# B&R Automation Studio project Teknologia25 (part 9)

#### BasicMovement.st
```iecst
ACTION BasicMoveDialGauge:
	pShuttle.function.MC_BR_MoveInPlane_Acp6D_0.Parameters.Acceleration := 5;
	pShuttle.function.MC_BR_MoveInPlane_Acp6D_0.Parameters.Velocity := 0.02;
	pShuttle.function.MC_BR_MoveInPlane_Acp6D_0.Shuttle := ADR(gAcp6DCtrl.Status.ShuttleInfo[pShuttle.par.shuttleID].shuttleRef);
	pShuttle.function.MC_BR_MoveInPlane_Acp6D_0.Parameters.Mode := 0; //Absolute
	pShuttle.function.MC_BR_MoveInPlane_Acp6D_0.Parameters.Path := 0; //direct

	CASE pShuttle.cm.state OF
		0:
			cm.description := 'Move shuttle to preDialPos';
			pShuttle.function.MC_BR_MoveInPlane_Acp6D_0.Parameters.Position.X := 0.420;
			pShuttle.function.MC_BR_MoveInPlane_Acp6D_0.Parameters.Position.Y := 0.180;
			pShuttle.function.MC_BR_MoveInPlane_Acp6D_0.Execute := TRUE;
			IF pShuttle.function.MC_BR_MoveInPlane_Acp6D_0.Acknowledge THEN
				pShuttle.function.MC_BR_MoveInPlane_Acp6D_0.Execute := FALSE;
				cm.state := 5;
			END_IF

		5:
			cm.description := 'Move shuttle to dialGauge';
			pShuttle.function.MC_BR_MoveInPlane_Acp6D_0.Parameters.Position.X := 0.420;
			pShuttle.function.MC_BR_MoveInPlane_Acp6D_0.Parameters.Position.Y := 0.190;
			pShuttle.function.MC_BR_MoveInPlane_Acp6D_0.Execute := TRUE;
			IF pShuttle.function.MC_BR_MoveInPlane_Acp6D_0.Acknowledge THEN
				pShuttle.function.MC_BR_MoveInPlane_Acp6D_0.Execute := FALSE;
				cm.state := 10;
			END_IF

		10:
			cm.description := 'Check pos reached';
			FOR i := 0 TO NUM_SHUTTLES DO
				IF((gAcp6DCtrl.Status.ShuttleInfo[pShuttle.par.shuttleID].Position.X > 0.420 - MARGIN AND gAcp6DCtrl.Status.ShuttleInfo[pShuttle.par.shuttleID].Position.X < 0.420 + MARGIN) AND
					gAcp6DCtrl.Status.ShuttleInfo[pShuttle.par.shuttleID].Position.Y > 0.190 - MARGIN AND gAcp6DCtrl.Status.ShuttleInfo[pShuttle.par.shuttleID].Position.Y < 0.190 + MARGIN) THEN
					IF gAcp6DCtrl.Status.ShuttleInfo[pShuttle.par.shuttleID].State = mcACP6D_SH_STATE_IDLING THEN
						cm.state := 20;
					END_IF
				END_IF
			END_FOR

		20:
			cm.description := 'Wait time';
			pShuttle.function.TON_0.PT := t#3s;
			pShuttle.function.TON_0.IN := TRUE;
			IF pShuttle.function.TON_0.Q THEN
				pShuttle.function.TON_0.IN := FALSE;
				cm.state := 30;
			END_IF

		30:
			cm.description := 'Move shuttle away from dialGauge';
			pShuttle.function.MC_BR_MoveInPlane_Acp6D_0.Parameters.Position.X := 0.420;
			pShuttle.function.MC_BR_MoveInPlane_Acp6D_0.Parameters.Position.Y := 0.180;
			pShuttle.function.MC_BR_MoveInPlane_Acp6D_0.Execute := TRUE;
			IF pShuttle.function.MC_BR_MoveInPlane_Acp6D_0.Acknowledge THEN
				pShuttle.function.MC_BR_MoveInPlane_Acp6D_0.Execute := FALSE;
				cm.state := 40;
			END_IF

		40:
			cm.description := 'Check pos reached';
			FOR i := 0 TO NUM_SHUTTLES DO
				IF((gAcp6DCtrl.Status.ShuttleInfo[pShuttle.par.shuttleID].Position.X > 0.420 - MARGIN AND gAcp6DCtrl.Status.ShuttleInfo[pShuttle.par.shuttleID].Position.X < 0.420 + MARGIN) AND
					gAcp6DCtrl.Status.ShuttleInfo[pShuttle.par.shuttleID].Position.Y > 0.180 - MARGIN AND gAcp6DCtrl.Status.ShuttleInfo[pShuttle.par.shuttleID].Position.Y < 0.180 + MARGIN) THEN
					IF gAcp6DCtrl.Status.ShuttleInfo[pShuttle.par.shuttleID].State = mcACP6D_SH_STATE_IDLING THEN
						cm.state := 0;
					END_IF
				END_IF
			END_FOR

	END_CASE

	cm();
	pShuttle.function.TON_0();
	pShuttle.function.MC_BR_MoveInPlane_Acp6D_0();

END_ACTION
```

#### WeightProgram.st
```iecst
ACTION weightProgram:
	pShuttle.function.MC_BR_ShGetPayload_Acp6D_0.Shuttle := ADR(gAcp6DCtrl.Status.ShuttleInfo[pShuttle.par.shuttleID].shuttleRef);

	pShuttle.function.MC_BR_MoveShortAxis_Acp6D_0.Shuttle := ADR(gAcp6DCtrl.Status.ShuttleInfo[pShuttle.par.shuttleID].shuttleRef);
	pShuttle.function.MC_BR_MoveShortAxis_Acp6D_0.Parameters.Position.Rx := 0.000;
	pShuttle.function.MC_BR_MoveShortAxis_Acp6D_0.Parameters.Position.Ry := 0.000;
	pShuttle.function.MC_BR_MoveShortAxis_Acp6D_0.Parameters.Position.Rz := 0.000;
	pShuttle.function.MC_BR_MoveShortAxis_Acp6D_0.Parameters.Position.Z := (weightProgramFlyingHight/1000); //mm to meter;
	pShuttle.function.MC_BR_MoveShortAxis_Acp6D_0.Parameters.Velocity.Z := 1;

	pShuttle.function.MC_BR_MoveInPlane_Acp6D_0.Shuttle := ADR(gAcp6DCtrl.Status.ShuttleInfo[pShuttle.par.shuttleID].shuttleRef);
	pShuttle.function.MC_BR_MoveInPlane_Acp6D_0.Parameters.Acceleration := 1;
	pShuttle.function.MC_BR_MoveInPlane_Acp6D_0.Parameters.Velocity := gAcp6DCtrl.Par.Velocity;
	pShuttle.function.MC_BR_MoveInPlane_Acp6D_0.Parameters.Path := 0; //Diagonal
	pShuttle.function.MC_BR_MoveInPlane_Acp6D_0.Parameters.Mode := 0; //absolute

	CASE cm.state OF
		0:
			cm.description := 'Move shuttle to loadLocation';
			pShuttle.function.MC_BR_MoveInPlane_Acp6D_0.Parameters.Position.X := 0.060;
			pShuttle.function.MC_BR_MoveInPlane_Acp6D_0.Parameters.Position.Y := 0.060;
			pShuttle.function.MC_BR_MoveInPlane_Acp6D_0.Execute := TRUE;
			IF pShuttle.function.MC_BR_MoveInPlane_Acp6D_0.Acknowledge THEN
				pShuttle.function.MC_BR_MoveInPlane_Acp6D_0.Execute := FALSE;
				cm.state := 5;
			END_IF

		5:
			cm.description := 'Change levitation hight';
			pShuttle.function.MC_BR_MoveShortAxis_Acp6D_0.Execute := TRUE;
			IF pShuttle.function.MC_BR_MoveShortAxis_Acp6D_0.Acknowledge THEN
				pShuttle.function.MC_BR_MoveShortAxis_Acp6D_0.Execute := FALSE;
				cm.state := 10;
			END_IF

		10:
			cm.description := 'Check pos reached';
			FOR i := 0 TO NUM_SHUTTLES DO
				IF((gAcp6DCtrl.Status.ShuttleInfo[pShuttle.par.shuttleID].Position.X > 0.060 - MARGIN AND gAcp6DCtrl.Status.ShuttleInfo[pShuttle.par.shuttleID].Position.X < 0.060 + MARGIN) AND
					gAcp6DCtrl.Status.ShuttleInfo[pShuttle.par.shuttleID].Position.Y > 0.060 - MARGIN AND gAcp6DCtrl.Status.ShuttleInfo[pShuttle.par.shuttleID].Position.Y < 0.060 + MARGIN) THEN
					IF gAcp6DCtrl.Status.ShuttleInfo[pShuttle.par.shuttleID].State = mcACP6D_SH_STATE_IDLING THEN
						cm.state := 20;
					END_IF
				END_IF
			END_FOR

		20:
			cm.description := 'Trigger robot';
			ABBRobot.startBigWeightMovement := TRUE;
			pShuttle.function.TON_0.PT := t#3s;
			pShuttle.function.TON_0.IN := TRUE;
			IF pShuttle.function.TON_0.Q THEN
				ABBRobot.startBigWeightMovement := FALSE;
				pShuttle.function.TON_0.IN := FALSE;
				cm.state := 21;
			END_IF

		21:
			cm.description := 'Calibrate weight';
			pShuttle.function.MC_BR_ShGetPayload_Acp6D_0.Execute := TRUE;
			IF pShuttle.function.MC_BR_ShGetPayload_Acp6D_0.Done THEN
				weightCalibration := pShuttle.function.MC_BR_ShGetPayload_Acp6D_0.Payload * 1000;
				pShuttle.function.MC_BR_ShGetPayload_Acp6D_0.Execute := FALSE;
				cm.state := 50;
			END_IF

//		25:
//			cm.description := 'Wait robot done';
//			IF ABBRobot.HomePositionReached THEN
//				cm.state := 50;
//			END_IF

		50:
			cm.description := 'Measure weight';
			pShuttle.function.MC_BR_ShGetPayload_Acp6D_0.Execute := TRUE;
			IF pShuttle.function.MC_BR_ShGetPayload_Acp6D_0.Done THEN
				fbPayload := pShuttle.function.MC_BR_ShGetPayload_Acp6D_0.Payload * 1000;
				shuttlePayload := fbPayload - weightCalibration;
				tempINT := REAL_TO_INT(shuttlePayload / 100);
				IF correctionValue = 0 THEN
					correctionValue := 12;
				END_IF;
				shuttlePayload := shuttlePayload - INT_TO_REAL(tempINT) * correctionValue;
				pShuttle.function.MC_BR_ShGetPayload_Acp6D_0.Execute := FALSE;
				cm.state := 60;
			END_IF

		60:
			cm.description := 'Wait time';
			pShuttle.function.TON_0.PT := t#1s;
			pShuttle.function.TON_0.IN := TRUE;
			IF pShuttle.function.TON_0.Q THEN
				pShuttle.function.TON_0.IN := FALSE;
				cm.state := 50;
			END_IF

//		80:
//			cm.description := 'Check robot ready';
//			IF ABBRobot.HomePositionReached THEN
//				ABBRobot.returnBigWeightMovement := TRUE;
//				cm.state := 81;
//			END_IF
//
//		81:
//			IF NOT ABBRobot.HomePositionReached THEN
//				ABBRobot.returnBigWeightMovement := FALSE;
//				cm.state := 90;
//			END_IF
//
//		90:
//			cm.description := 'Check when robot is done and fire small weightMovement';
//			IF ABBRobot.HomePositionReached THEN
//				ABBRobot.startSmallWeightMovement := TRUE;
//				cm.state := 100;
//			END_IF
//
//		100:
//			cm.description := 'Check robot start';
//			IF NOT ABBRobot.HomePositionReached THEN
//				ABBRobot.startSmallWeightMovement := FALSE;
//				cm.state := 110;
//			END_IF
//
//		110:
//			cm.description := 'Check robot done';
//			IF ABBRobot.HomePositionReached THEN
//				cm.state := 120;
//			END_IF
//
//		120:
//			cm.description := 'meassure small weight';
//			pShuttle.function.MC_BR_GetPayload_Acp6D_0.Execute := TRUE;
//			IF pShuttle.function.MC_BR_GetPayload_Acp6D_0.Valid THEN
//				shuttlePayload := pShuttle.function.MC_BR_GetPayload_Acp6D_0.Payload * 1000;
//				shuttlePayload := shuttlePayload - weightCalibration;
//				pShuttle.function.MC_BR_GetPayload_Acp6D_0.Execute := FALSE;
//				cm.state := 130;
//			END_IF
//
//		130:
//			cm.description := 'Wait time';
//			pShuttle.function.TON_0.PT := t#3s;
//			pShuttle.function.TON_0.IN := TRUE;
//			IF pShuttle.function.TON_0.Q THEN
//				pShuttle.function.TON_0.IN := FALSE;
//				cm.state := 140;
//			END_IF
//
//		140:
//			cm.description := 'Return small weight';
//			IF ABBRobot.HomePositionReached THEN
//				ABBRobot.returnSmallWeightMovement := TRUE;
//				cm.state := 150;
//			END_IF
//
//		150:
//			IF NOT ABBRobot.HomePositionReached THEN
//				ABBRobot.returnSmallWeightMovement := FALSE;
//				cm.state := 160;
//			END_IF
//
//		160:
//			IF ABBRobot.HomePositionReached THEN
//				modeSelector := 5; //demoProgram
//				em.cmd.sc := TRUE;
//			END_IF

	END_CASE
	pShuttle.function.MC_BR_MoveShortAxis_Acp6D_0();
	pShuttle.function.MC_BR_ShGetPayload_Acp6D_0();
	pShuttle.function.MC_BR_MoveInPlane_Acp6D_0();
	pShuttle.function.TON_0();
END_ACTION
```

#### MovementRxRyRz.st
```iecst
ACTION MovementRx:
	pShuttle.function.MC_BR_MoveShortAxis_Acp6D_0.Shuttle := ADR(gAcp6DCtrl.Status.ShuttleInfo[pShuttle.par.shuttleID].shuttleRef);
	pShuttle.function.MC_BR_MoveShortAxis_Acp6D_0.Parameters.Mode := 0; //Absolute
	pShuttle.function.MC_BR_MoveShortAxis_Acp6D_0.Parameters.Rotation.Type := 0; //Around Center
	pShuttle.function.MC_BR_MoveShortAxis_Acp6D_0.Parameters.Velocity.Rx := 0.1;
	pShuttle.function.MC_BR_MoveShortAxis_Acp6D_0.Parameters.Velocity.Rx := 0.1;
	pShuttle.function.MC_BR_MoveShortAxis_Acp6D_0.Parameters.Velocity.Ry := 0.1;
	pShuttle.function.MC_BR_MoveShortAxis_Acp6D_0.Parameters.Velocity.Z := 0.002;

	pShuttle.function.MC_BR_Move6D_Acp6D_0.Shuttle := ADR(gAcp6DCtrl.Status.ShuttleInfo[pShuttle.par.shuttleID].shuttleRef);
	CASE cm.state OF
		0:
			cm.description := 'tilt shuttle Rx';
			pShuttle.function.MC_BR_MoveShortAxis_Acp6D_0.Parameters.Position.Z := 0.002;
			pShuttle.function.MC_BR_MoveShortAxis_Acp6D_0.Parameters.Position.Rx := 0.02;
			pShuttle.function.MC_BR_MoveShortAxis_Acp6D_0.Parameters.Position.Ry := 0.00;
			pShuttle.function.MC_BR_MoveShortAxis_Acp6D_0.Parameters.Position.Rz := 0.00;
			pShuttle.function.MC_BR_MoveShortAxis_Acp6D_0.Execute := TRUE;
			IF pShuttle.function.MC_BR_MoveShortAxis_Acp6D_0.Acknowledge THEN
				pShuttle.function.MC_BR_MoveShortAxis_Acp6D_0.Execute := FALSE;
				cm.state := 10;
			ELSIF pShuttle.function.MC_BR_MoveShortAxis_Acp6D_0.Error THEN
				em.cmd.abort := TRUE;
			END_IF;

		10:
			cm.description := 'Check Rx position reached';
			IF gAcp6DCtrl.Status.ShuttleInfo[pShuttle.par.shuttleID].Position.Rx >= 0.019 THEN
				cm.state := 20;
			END_IF

		20:
			cm.description := 'tilt shuttle Rx';
			pShuttle.function.MC_BR_MoveShortAxis_Acp6D_0.Parameters.Position.Z := 0.002;
			pShuttle.function.MC_BR_MoveShortAxis_Acp6D_0.Parameters.Position.Rx := -0.02;
			pShuttle.function.MC_BR_MoveShortAxis_Acp6D_0.Parameters.Position.Ry := 0.00;
			pShuttle.function.MC_BR_MoveShortAxis_Acp6D_0.Parameters.Position.Rz := 0.00;
			pShuttle.function.MC_BR_MoveShortAxis_Acp6D_0.Execute := TRUE;
			IF pShuttle.function.MC_BR_MoveShortAxis_Acp6D_0.Acknowledge THEN
				pShuttle.function.MC_BR_MoveShortAxis_Acp6D_0.Execute := FALSE;
				cm.state := 30;
			ELSIF pShuttle.function.MC_BR_MoveShortAxis_Acp6D_0.Error THEN
				em.cmd.abort := TRUE;
			END_IF;

		30:
			cm.description := 'Check Rx position reached';
			IF gAcp6DCtrl.Status.ShuttleInfo[pShuttle.par.shuttleID].Position.Rx <= -0.019 THEN
				cm.state := 0;
			END_IF

	END_CASE

	cm();
	pShuttle.function.MC_BR_MoveShortAxis_Acp6D_0();
	pShuttle.function.MC_BR_Move6D_Acp6D_0();

END_ACTION

ACTION MovementRy:
	pShuttle.function.MC_BR_MoveShortAxis_Acp6D_0.Shuttle := ADR(gAcp6DCtrl.Status.ShuttleInfo[pShuttle.par.shuttleID].shuttleRef);
	pShuttle.function.MC_BR_MoveShortAxis_Acp6D_0.Parameters.Mode := 0; //Absolute
	pShuttle.function.MC_BR_MoveShortAxis_Acp6D_0.Parameters.Rotation.Type := 0; //Around Center
	pShuttle.function.MC_BR_MoveShortAxis_Acp6D_0.Parameters.Velocity.Rx := 0.1;
	pShuttle.function.MC_BR_MoveShortAxis_Acp6D_0.Parameters.Velocity.Rx := 0.1;
	pShuttle.function.MC_BR_MoveShortAxis_Acp6D_0.Parameters.Velocity.Ry := 0.1;
	pShuttle.function.MC_BR_MoveShortAxis_Acp6D_0.Parameters.Velocity.Z := 0.002;

	pShuttle.function.MC_BR_Move6D_Acp6D_0.Shuttle := ADR(gAcp6DCtrl.Status.ShuttleInfo[pShuttle.par.shuttleID].shuttleRef);

	CASE cm.state OF
		0:

			cm.description := 'tilt shuttle Ry';
			pShuttle.function.MC_BR_MoveShortAxis_Acp6D_0.Parameters.Position.Z := 0.002;
			pShuttle.function.MC_BR_MoveShortAxis_Acp6D_0.Parameters.Position.Ry := 0.02;
			pShuttle.function.MC_BR_MoveShortAxis_Acp6D_0.Parameters.Position.Rx := 0.00;
			pShuttle.function.MC_BR_MoveShortAxis_Acp6D_0.Parameters.Position.Rz := 0.00;
			pShuttle.function.MC_BR_MoveShortAxis_Acp6D_0.Execute := TRUE;
			IF pShuttle.function.MC_BR_MoveShortAxis_Acp6D_0.Acknowledge THEN
				pShuttle.function.MC_BR_MoveShortAxis_Acp6D_0.Execute := FALSE;
				cm.state := 10;
			ELSIF pShuttle.function.MC_BR_MoveShortAxis_Acp6D_0.Error THEN
				em.cmd.abort := TRUE;
			END_IF;

		10:
			cm.description := 'Check Rx position reached';
			IF gAcp6DCtrl.Status.ShuttleInfo[pShuttle.par.shuttleID].Position.Ry >= 0.019 THEN
				cm.state := 20;
			END_IF

		20:
			cm.description := 'tilt shuttle Ry';
			pShuttle.function.MC_BR_MoveShortAxis_Acp6D_0.Parameters.Position.Z := 0.002;
			pShuttle.function.MC_BR_MoveShortAxis_Acp6D_0.Parameters.Position.Ry := -0.02;
			pShuttle.function.MC_BR_MoveShortAxis_Acp6D_0.Parameters.Position.Rx := 0.00;
			pShuttle.function.MC_BR_MoveShortAxis_Acp6D_0.Parameters.Position.Rz := 0.00;
			pShuttle.function.MC_BR_MoveShortAxis_Acp6D_0.Execute := TRUE;
			IF pShuttle.function.MC_BR_MoveShortAxis_Acp6D_0.Acknowledge THEN
				pShuttle.function.MC_BR_MoveShortAxis_Acp6D_0.Execute := FALSE;
				cm.state := 30;
			ELSIF pShuttle.function.MC_BR_MoveShortAxis_Acp6D_0.Error THEN
				em.cmd.abort := TRUE;
			END_IF;

		30:
			cm.description := 'Check Ry position reached';
			IF gAcp6DCtrl.Status.ShuttleInfo[pShuttle.par.shuttleID].Position.Ry <= -0.019 THEN
				cm.state := 0;
			END_IF

	END_CASE

	cm();
	pShuttle.function.MC_BR_MoveShortAxis_Acp6D_0();
	pShuttle.function.MC_BR_Move6D_Acp6D_0();

END_ACTION

ACTION MovementRz:
	pShuttle.function.MC_BR_MoveShortAxis_Acp6D_0.Shuttle := ADR(gAcp6DCtrl.Status.ShuttleInfo[pShuttle.par.shuttleID].shuttleRef);
	pShuttle.function.MC_BR_MoveShortAxis_Acp6D_0.Parameters.Mode := 0; //Absolute
	pShuttle.function.MC_BR_MoveShortAxis_Acp6D_0.Parameters.Rotation.Type := 0; //Around Center
	pShuttle.function.MC_BR_MoveShortAxis_Acp6D_0.Parameters.Velocity.Rx := 0.1;
	pShuttle.function.MC_BR_MoveShortAxis_Acp6D_0.Parameters.Velocity.Rx := 0.1;
	pShuttle.function.MC_BR_MoveShortAxis_Acp6D_0.Parameters.Velocity.Ry := 0.1;
	pShuttle.function.MC_BR_MoveShortAxis_Acp6D_0.Parameters.Velocity.Z := 0.002;

	pShuttle.function.MC_BR_Move6D_Acp6D_0.Shuttle := ADR(gAcp6DCtrl.Status.ShuttleInfo[pShuttle.par.shuttleID].shuttleRef);
	CASE cm.state OF
		0:

			cm.description := 'tilt shuttle Rz';
			pShuttle.function.MC_BR_MoveShortAxis_Acp6D_0.Parameters.Position.Z := 0.002;
			pShuttle.function.MC_BR_MoveShortAxis_Acp6D_0.Parameters.Position.Rz := 0.150;
			pShuttle.function.MC_BR_MoveShortAxis_Acp6D_0.Parameters.Position.Rx := 0.00;
			pShuttle.function.MC_BR_MoveShortAxis_Acp6D_0.Parameters.Position.Ry := 0.00;
			pShuttle.function.MC_BR_MoveShortAxis_Acp6D_0.Execute := TRUE;
			IF pShuttle.function.MC_BR_MoveShortAxis_Acp6D_0.Acknowledge THEN
				pShuttle.function.MC_BR_MoveShortAxis_Acp6D_0.Execute := FALSE;
				cm.state := 10;
			ELSIF pShuttle.function.MC_BR_MoveShortAxis_Acp6D_0.Error THEN
				em.cmd.abort := TRUE;
			END_IF;

		10:
			cm.description := 'Check Rx position reached';
			IF gAcp6DCtrl.Status.ShuttleInfo[pShuttle.par.shuttleID].Position.RZ >= 0.0140 THEN
				cm.state := 20;
			END_IF

		20:
			cm.description := 'tilt shuttle Rz';
			pShuttle.function.MC_BR_MoveShortAxis_Acp6D_0.Parameters.Position.Z := 0.002;
			pShuttle.function.MC_BR_MoveShortAxis_Acp6D_0.Parameters.Position.Rz := -0.150;
			pShuttle.function.MC_BR_MoveShortAxis_Acp6D_0.Parameters.Position.Rx := 0.00;
			pShuttle.function.MC_BR_MoveShortAxis_Acp6D_0.Parameters.Position.Ry := 0.00;
			pShuttle.function.MC_BR_MoveShortAxis_Acp6D_0.Execute := TRUE;
			IF pShuttle.function.MC_BR_MoveShortAxis_Acp6D_0.Acknowledge THEN
				pShuttle.function.MC_BR_MoveShortAxis_Acp6D_0.Execute := FALSE;
				cm.state := 30;
			ELSIF pShuttle.function.MC_BR_MoveShortAxis_Acp6D_0.Aborted THEN
				em.cmd.abort := TRUE;
			END_IF;

		30:
			cm.description := 'Check Rx position reached';
			IF gAcp6DCtrl.Status.ShuttleInfo[pShuttle.par.shuttleID].Position.RZ <= -0.0140 THEN
				cm.state := 0;
			END_IF

	END_CASE

	cm();
	pShuttle.function.MC_BR_MoveShortAxis_Acp6D_0();
	pShuttle.function.MC_BR_Move6D_Acp6D_0();

END_ACTION

ACTION MovementZ:
	pShuttle.function.MC_BR_MoveShortAxis_Acp6D_0.Shuttle := ADR(gAcp6DCtrl.Status.ShuttleInfo[pShuttle.par.shuttleID].shuttleRef);
	pShuttle.function.MC_BR_MoveShortAxis_Acp6D_0.Parameters.Mode := 0; //Absolute
	pShuttle.function.MC_BR_MoveShortAxis_Acp6D_0.Parameters.Rotation.Type := 0; //Around Center
	pShuttle.function.MC_BR_MoveShortAxis_Acp6D_0.Parameters.Velocity.Rx := 0.1;
	pShuttle.function.MC_BR_MoveShortAxis_Acp6D_0.Parameters.Velocity.Rx := 0.1;
	pShuttle.function.MC_BR_MoveShortAxis_Acp6D_0.Parameters.Velocity.Ry := 0.1;
	pShuttle.function.MC_BR_MoveShortAxis_Acp6D_0.Parameters.Velocity.Z := 0.002;
	CASE em.substate OF
//		12000..12999:
//			pShuttle.function.MC_BR_MoveShortAxis_Acp6D_0.Parameters.Velocity.Z := 2;
		ELSE
			//pShuttle.function.MC_BR_MoveShortAxis_Acp6D_0.Parameters.Velocity.Z := 0.002;
			pShuttle.function.MC_BR_MoveShortAxis_Acp6D_0.Parameters.Velocity.Z := levitationVelocity;
	END_CASE
	pShuttle.function.MC_BR_Move6D_Acp6D_0.Shuttle := ADR(gAcp6DCtrl.Status.ShuttleInfo[pShuttle.par.shuttleID].shuttleRef);

	CASE cm.state OF
		0:

			cm.description := 'raise shuttle';
			pShuttle.function.MC_BR_MoveShortAxis_Acp6D_0.Parameters.Position.Z := 0.004;
			pShuttle.function.MC_BR_MoveShortAxis_Acp6D_0.Parameters.Position.Rz := 0.00;
			pShuttle.function.MC_BR_MoveShortAxis_Acp6D_0.Parameters.Position.Rx := 0.00;
			pShuttle.function.MC_BR_MoveShortAxis_Acp6D_0.Parameters.Position.Ry := 0.00;
			pShuttle.function.MC_BR_MoveShortAxis_Acp6D_0.Execute := TRUE;
			IF pShuttle.function.MC_BR_MoveShortAxis_Acp6D_0.Acknowledge THEN
				pShuttle.function.MC_BR_MoveShortAxis_Acp6D_0.Execute := FALSE;
				cm.state := 10;
			ELSIF pShuttle.function.MC_BR_MoveShortAxis_Acp6D_0.Error THEN
				em.cmd.abort := TRUE;
			END_IF;

		10:
			cm.description := 'Check Rx position reached';
			IF gAcp6DCtrl.Status.ShuttleInfo[pShuttle.par.shuttleID].Position.Z >= 0.0038 THEN
				cm.state := 20;
			END_IF

		20:
			cm.description := 'tilt shuttle Rz';
			pShuttle.function.MC_BR_MoveShortAxis_Acp6D_0.Parameters.Position.Z := 0.001;
			pShuttle.function.MC_BR_MoveShortAxis_Acp6D_0.Parameters.Position.Rz := 0.00;
			pShuttle.function.MC_BR_MoveShortAxis_Acp6D_0.Parameters.Position.Rx := 0.00;
			pShuttle.function.MC_BR_MoveShortAxis_Acp6D_0.Parameters.Position.Ry := 0.00;
			pShuttle.function.MC_BR_MoveShortAxis_Acp6D_0.Execute := TRUE;
			IF pShuttle.function.MC_BR_MoveShortAxis_Acp6D_0.Acknowledge THEN
				pShuttle.function.MC_BR_MoveShortAxis_Acp6D_0.Execute := FALSE;
				cm.state := 30;
			ELSIF pShuttle.function.MC_BR_MoveShortAxis_Acp6D_0.Error THEN
				em.cmd.abort := TRUE;
			END_IF;

		30:
			cm.description := 'Check Rz position reached';
			IF gAcp6DCtrl.Status.ShuttleInfo[pShuttle.par.shuttleID].Position.Z <= 0.0011 THEN
				cm.state := 0;
			END_IF

	END_CASE

	cm();
	pShuttle.function.MC_BR_MoveShortAxis_Acp6D_0();
	pShuttle.function.MC_BR_Move6D_Acp6D_0();
END_ACTION
```

#### linkMovement.st
```iecst
ACTION linkMovementProgram:
	//Setup
	positionContainerLinkMovement[0].Shuttle1.xPos := 0.120;
	positionContainerLinkMovement[0].Shuttle1.yPos := 0.120;
	positionContainerLinkMovement[0].Shuttle2.xPos := 0.360;
	positionContainerLinkMovement[0].Shuttle2.yPos := 0.360;
	positionContainerLinkMovement[0].Shuttle3.xPos := 0.360;
	positionContainerLinkMovement[0].Shuttle3.yPos := 0.120;
	positionContainerLinkMovement[0].Shuttle4.xPos := 0.120;
	positionContainerLinkMovement[0].Shuttle4.yPos := 0.360;

	positionContainerLinkMovement[1].Shuttle1.xPos := 0.060;
	positionContainerLinkMovement[1].Shuttle1.yPos := 0.060;
	positionContainerLinkMovement[1].Shuttle2.xPos := 0.180;
	positionContainerLinkMovement[1].Shuttle2.yPos := 0.180;
	positionContainerLinkMovement[1].Shuttle3.xPos := 0.180;
	positionContainerLinkMovement[1].Shuttle3.yPos := 0.060;
	positionContainerLinkMovement[1].Shuttle4.xPos := 0.060;
	positionContainerLinkMovement[1].Shuttle4.yPos := 0.180;

	positionContainerLinkMovement[2].Shuttle1.xPos := 0.120;
	positionContainerLinkMovement[2].Shuttle1.yPos := 0.120;
	positionContainerLinkMovement[2].Shuttle2.xPos := 0.360;
	positionContainerLinkMovement[2].Shuttle2.yPos := 0.360;
	positionContainerLinkMovement[2].Shuttle3.xPos := 0.360;
	positionContainerLinkMovement[2].Shuttle3.yPos := 0.120;
	positionContainerLinkMovement[2].Shuttle4.xPos := 0.120;
	positionContainerLinkMovement[2].Shuttle4.yPos := 0.360;

	positionContainerLinkMovement[3].Shuttle1.xPos := 0.300;
	positionContainerLinkMovement[3].Shuttle1.yPos := 0.060;
	positionContainerLinkMovement[3].Shuttle2.xPos := 0.420;
	positionContainerLinkMovement[3].Shuttle2.yPos := 0.180;
	positionContainerLinkMovement[3].Shuttle3.xPos := 0.420;
	positionContainerLinkMovement[3].Shuttle3.yPos := 0.060;
	positionContainerLinkMovement[3].Shuttle4.xPos := 0.300;
	positionContainerLinkMovement[3].Shuttle4.yPos := 0.180;

	positionContainerLinkMovement[4].Shuttle1.xPos := 0.120;
	positionContainerLinkMovement[4].Shuttle1.yPos := 0.120;
	positionContainerLinkMovement[4].Shuttle2.xPos := 0.360;
	positionContainerLinkMovement[4].Shuttle2.yPos := 0.360;
	positionContainerLinkMovement[4].Shuttle3.xPos := 0.360;
	positionContainerLinkMovement[4].Shuttle3.yPos := 0.120;
	positionContainerLinkMovement[4].Shuttle4.xPos := 0.120;
	positionContainerLinkMovement[4].Shuttle4.yPos := 0.360;

	positionContainerLinkMovement[5].Shuttle1.xPos := 0.300;
	positionContainerLinkMovement[5].Shuttle1.yPos := 0.300;
	positionContainerLinkMovement[5].Shuttle2.xPos := 0.420;
	positionContainerLinkMovement[5].Shuttle2.yPos := 0.420;
	positionContainerLinkMovement[5].Shuttle3.xPos := 0.420;
	positionContainerLinkMovement[5].Shuttle3.yPos := 0.300;
	positionContainerLinkMovement[5].Shuttle4.xPos := 0.300;
	positionContainerLinkMovement[5].Shuttle4.yPos := 0.420;

	positionContainerLinkMovement[6].Shuttle1.xPos := 0.120;
	positionContainerLinkMovement[6].Shuttle1.yPos := 0.120;
	positionContainerLinkMovement[6].Shuttle2.xPos := 0.360;
	positionContainerLinkMovement[6].Shuttle2.yPos := 0.360;
	positionContainerLinkMovement[6].Shuttle3.xPos := 0.360;
	positionContainerLinkMovement[6].Shuttle3.yPos := 0.120;
	positionContainerLinkMovement[6].Shuttle4.xPos := 0.120;
	positionContainerLinkMovement[6].Shuttle4.yPos := 0.360;

	CASE em.substate OF
		3000:
			em.description := 'Move all shuttles to prePos';
			tempShuttleCounter := 0;
			tempCounter := 0;
			em.substate := 3010;

		3010:
			em.description := 'Move all shuttles to prePos';
			IF tempShuttleCounter > NUM_SHUTTLES THEN
				tempShuttleCounter := 0;
				em.substate := 3030;
			ELSE
				MC_BR_MoveInPlane_Acp6D_0.Parameters.Acceleration := gAcp6DCtrl.Par.Acceleration;
				MC_BR_MoveInPlane_Acp6D_0.Parameters.Velocity := gAcp6DCtrl.Par.Velocity;
				MC_BR_MoveInPlane_Acp6D_0.Parameters.Mode := 0; //Abs
				MC_BR_MoveInPlane_Acp6D_0.Shuttle := ADR(gAcp6DCtrl.Status.ShuttleInfo[tempShuttleCounter].shuttleRef);
				CASE tempShuttleCounter OF
					0:
						MC_BR_MoveInPlane_Acp6D_0.Parameters.Position.X := 0.060;
						MC_BR_MoveInPlane_Acp6D_0.Parameters.Position.Y := 0.180;
					1:
						MC_BR_MoveInPlane_Acp6D_0.Parameters.Position.X := 0.180;
						MC_BR_MoveInPlane_Acp6D_0.Parameters.Position.Y := 0.180;
					2:
						MC_BR_MoveInPlane_Acp6D_0.Parameters.Position.X := 0.300;
						MC_BR_MoveInPlane_Acp6D_0.Parameters.Position.Y := 0.060;
					3:
						MC_BR_MoveInPlane_Acp6D_0.Parameters.Position.X := 0.420;
						MC_BR_MoveInPlane_Acp6D_0.Parameters.Position.Y := 0.060;
				END_CASE

				MC_BR_MoveInPlane_Acp6D_0.Execute := TRUE;
				IF MC_BR_MoveInPlane_Acp6D_0.Acknowledge THEN
					MC_BR_MoveInPlane_Acp6D_0.Execute := FALSE;
					tempShuttleCounter := tempShuttleCounter + 1;
					em.substate := 3020;
				END_IF
			END_IF

		3020:
			em.description := 'DummyScan';
			em.substate := 3010;

		3030:
			em.description := 'check shuttle state idle';
			IF gAcp6DCtrl.Status.ShuttleInfo[0].State = mcACP6D_SH_STATE_IDLING AND gAcp6DCtrl.Status.ShuttleInfo[1].State = mcACP6D_SH_STATE_IDLING
				AND gAcp6DCtrl.Status.ShuttleInfo[2].State = mcACP6D_SH_STATE_IDLING AND gAcp6DCtrl.Status.ShuttleInfo[3].State = mcACP6D_SH_STATE_IDLING AND MC_BR_AsmReadStatus_Acp6D_0.AssemblyReady THEN
				em.substate := 3035;
			END_IF

		3035:
			em.description := 'Couple ShuttleGroup1_2';
			em.cmd.sc := FALSE;
			MC_BR_ShGroupCoupleCtrl_Acp6D_0.ShuttleGroup := shGroupShuttle1_2;
			MC_BR_ShGroupCoupleCtrl_Acp6D_0.Parameters.Option := 1; //Couple
			MC_BR_ShGroupCoupleCtrl_Acp6D_0.Execute := TRUE;
			IF MC_BR_ShGroupCoupleCtrl_Acp6D_0.Done THEN
				MC_BR_ShGroupCoupleCtrl_Acp6D_0.Execute := FALSE;
				em.substate := 3040;
			ELSIF MC_BR_ShGroupCoupleCtrl_Acp6D_0.Error THEN
				em.cmd.abort := TRUE;
			END_IF

		3040:
			em.description := 'Couple ShuttleGroup1_2';
			em.cmd.sc := FALSE;
			MC_BR_ShGroupCoupleCtrl_Acp6D_0.ShuttleGroup := shGroupShuttle3_4;
			MC_BR_ShGroupCoupleCtrl_Acp6D_0.Parameters.Option := 1; //Couple
			MC_BR_ShGroupCoupleCtrl_Acp6D_0.Execute := TRUE;
			IF MC_BR_ShGroupCoupleCtrl_Acp6D_0.Done THEN
				MC_BR_ShGroupCoupleCtrl_Acp6D_0.Execute := FALSE;
				em.substate := 3050;
			ELSIF MC_BR_ShGroupCoupleCtrl_Acp6D_0.Error THEN
				em.cmd.abort := TRUE;
			END_IF

		3050:
			em.description := 'Move group 10 of shuttle around';
			em.cmd.sc := FALSE;
			IF tempCounter >= 3 THEN
				tempCounter := 0;
				em.substate := 3070;
			ELSE
				MC_BR_MoveInPlane_Acp6D_0.Shuttle := ADR(gAcp6DCtrl.Status.ShuttleInfo[0].shuttleRef);
				MC_BR_MoveInPlane_Acp6D_0.Parameters.Position.X := 0.300;
				MC_BR_MoveInPlane_Acp6D_0.Parameters.Position.Y := 0.060;
				MC_BR_MoveInPlane_Acp6D_0.Parameters.Path := 2; //Y then X
				MC_BR_MoveInPlane_Acp6D_0.Execute := TRUE;
				IF MC_BR_MoveInPlane_Acp6D_0.Acknowledge THEN
					MC_BR_MoveInPlane_Acp6D_0.Execute := FALSE;
					em.substate := 3060;
				END_IF
			END_IF

		3060:
			em.description := 'Move group of shuttle around';
			em.cmd.sc := FALSE;
			MC_BR_MoveInPlane_Acp6D_0.Shuttle := ADR(gAcp6DCtrl.Status.ShuttleInfo[0].shuttleRef);
			MC_BR_MoveInPlane_Acp6D_0.Parameters.Position.X := 0.060;
			MC_BR_MoveInPlane_Acp6D_0.Parameters.Velocity := gAcp6DCtrl.Par.Velocity;
			MC_BR_MoveInPlane_Acp6D_0.Parameters.Acceleration := gAcp6DCtrl.Par.Acceleration;
			MC_BR_MoveInPlane_Acp6D_0.Parameters.Position.Y := 0.180;
			MC_BR_MoveInPlane_Acp6D_0.Parameters.Path := 2; //Y then X
			MC_BR_MoveInPlane_Acp6D_0.Execute := TRUE;
			IF MC_BR_MoveInPlane_Acp6D_0.Acknowledge THEN
				MC_BR_MoveInPlane_Acp6D_0.Execute := FALSE;
				tempCounter := tempCounter + 1;
				em.substate := 3050;
			END_IF

		3070:
			em.description := 'Move group 11 of shuttle around';
			em.cmd.sc := FALSE;
			IF tempCounter >= 3 THEN
				tempCounter := 0;
				em.substate := 3090;
			ELSE
				MC_BR_MoveInPlane_Acp6D_0.Shuttle := ADR(gAcp6DCtrl.Status.ShuttleInfo[2].shuttleRef);
				MC_BR_MoveInPlane_Acp6D_0.Parameters.Position.X := 0.060;
				MC_BR_MoveInPlane_Acp6D_0.Parameters.Position.Y := 0.180;
				MC_BR_MoveInPlane_Acp6D_0.Parameters.Path := 2; //Y then X
				MC_BR_MoveInPlane_Acp6D_0.Execute := TRUE;
				IF MC_BR_MoveInPlane_Acp6D_0.Acknowledge THEN
					MC_BR_MoveInPlane_Acp6D_0.Execute := FALSE;
					em.substate := 3080;
				END_IF
			END_IF

		3080:
			em.description := 'Move group of shuttle around';
			em.cmd.sc := FALSE;
			MC_BR_MoveInPlane_Acp6D_0.Shuttle := ADR(gAcp6DCtrl.Status.ShuttleInfo[2].shuttleRef);
			MC_BR_MoveInPlane_Acp6D_0.Parameters.Position.X := 0.300;
			MC_BR_MoveInPlane_Acp6D_0.Parameters.Velocity := gAcp6DCtrl.Par.Velocity;
			MC_BR_MoveInPlane_Acp6D_0.Parameters.Acceleration := gAcp6DCtrl.Par.Acceleration;
			MC_BR_MoveInPlane_Acp6D_0.Parameters.Position.Y := 0.060;
			MC_BR_MoveInPlane_Acp6D_0.Parameters.Path := 2; //Y then X
			MC_BR_MoveInPlane_Acp6D_0.Execute := TRUE;
			IF MC_BR_MoveInPlane_Acp6D_0.Acknowledge THEN
				MC_BR_MoveInPlane_Acp6D_0.Execute := FALSE;
				tempCounter := tempCounter + 1;
				em.substate := 3070;
			END_IF

		3090:
			em.description := 'DeCouple ShuttleGroup1_2';
			em.cmd.sc := FALSE;
			MC_BR_ShGroupCoupleCtrl_Acp6D_0.ShuttleGroup := shGroupShuttle1_2;
			MC_BR_ShGroupCoupleCtrl_Acp6D_0.Parameters.Option := 0; //DeCouple
			MC_BR_ShGroupCoupleCtrl_Acp6D_0.Execute := TRUE;
			IF MC_BR_ShGroupCoupleCtrl_Acp6D_0.Done THEN
				MC_BR_ShGroupCoupleCtrl_Acp6D_0.Execute := FALSE;
				em.substate := 3100;
			ELSIF MC_BR_ShGroupCoupleCtrl_Acp6D_0.Error THEN
				em.cmd.abort := TRUE;
			END_IF

		3100:
			em.description := 'Wait for shuttle to reach pos';
			em.cmd.sc := FALSE;
			IF((gAcp6DCtrl.Status.ShuttleInfo[2].Position.X > 0.300 - MARGIN AND gAcp6DCtrl.Status.ShuttleInfo[2].Position.X < 0.300 + MARGIN) AND
				gAcp6DCtrl.Status.ShuttleInfo[2].Position.Y > 0.060 - MARGIN AND gAcp6DCtrl.Status.ShuttleInfo[2].Position.Y < 0.060 + MARGIN) THEN
				IF gAcp6DCtrl.Status.ShuttleInfo[2].State = mcACP6D_SH_STATE_IDLING THEN
					em.substate := 3110;
				END_IF
			END_IF

		3110:
			em.description := 'Move right group up';
			em.cmd.sc := FALSE;
			MC_BR_MoveInPlane_Acp6D_0.Shuttle := ADR(gAcp6DCtrl.Status.ShuttleInfo[2].shuttleRef);
			MC_BR_MoveInPlane_Acp6D_0.Parameters.Position.X := 0.300;
			MC_BR_MoveInPlane_Acp6D_0.Parameters.Velocity := gAcp6DCtrl.Par.Velocity;
			MC_BR_MoveInPlane_Acp6D_0.Parameters.Acceleration := gAcp6DCtrl.Par.Acceleration;
			MC_BR_MoveInPlane_Acp6D_0.Parameters.Position.Y := 0.180;
			MC_BR_MoveInPlane_Acp6D_0.Parameters.Path := 0; //Direct
			MC_BR_MoveInPlane_Acp6D_0.Execute := TRUE;
			IF MC_BR_MoveInPlane_Acp6D_0.Acknowledge THEN
				MC_BR_MoveInPlane_Acp6D_0.Execute := FALSE;
				em.substate := 3120;
			END_IF

		3120:
			em.description := 'Couple ShuttleGroup1_2';
			em.cmd.sc := FALSE;
			MC_BR_ShGroupCoupleCtrl_Acp6D_0.ShuttleGroup := shGroupShuttle3_4;
			MC_BR_ShGroupCoupleCtrl_Acp6D_0.Parameters.Option := 0; //DeCouple
			MC_BR_ShGroupCoupleCtrl_Acp6D_0.Execute := TRUE;
			IF MC_BR_ShGroupCoupleCtrl_Acp6D_0.Done THEN
				MC_BR_ShGroupCoupleCtrl_Acp6D_0.Execute := FALSE;
				em.substate := 3130;
			ELSIF MC_BR_ShGroupCoupleCtrl_Acp6D_0.Error THEN
				em.cmd.abort := TRUE;
			END_IF

		3130:
			em.description := 'rotationMove part 1';
			MC_BR_MoveInPlane_Acp6D_0.Shuttle := ADR(gAcp6DCtrl.Status.ShuttleInfo[1].shuttleRef);
			MC_BR_MoveInPlane_Acp6D_0.Parameters.Position.X := 0.060;
			MC_BR_MoveInPlane_Acp6D_0.Parameters.Velocity := gAcp6DCtrl.Par.Velocity;
			MC_BR_MoveInPlane_Acp6D_0.Parameters.Acceleration := gAcp6DCtrl.Par.Acceleration;
			MC_BR_MoveInPlane_Acp6D_0.Parameters.Position.Y := 0.060;
			MC_BR_MoveInPlane_Acp6D_0.Parameters.Path := 2; //Y then X
			MC_BR_MoveInPlane_Acp6D_0.Execute := TRUE;
			IF MC_BR_MoveInPlane_Acp6D_0.Acknowledge THEN
				MC_BR_MoveInPlane_Acp6D_0.Execute := FALSE;
				em.substate := 3140;
			END_IF

		3140:
			em.description := 'rotationMove part 2';
			MC_BR_MoveInPlane_Acp6D_0.Shuttle := ADR(gAcp6DCtrl.Status.ShuttleInfo[3].shuttleRef);
			MC_BR_MoveInPlane_Acp6D_0.Parameters.Position.X := 0.180;
			MC_BR_MoveInPlane_Acp6D_0.Parameters.Velocity := gAcp6DCtrl.Par.Velocity;
			MC_BR_MoveInPlane_Acp6D_0.Parameters.Acceleration := gAcp6DCtrl.Par.Acceleration;
			MC_BR_MoveInPlane_Acp6D_0.Parameters.Position.Y := 0.060;
			MC_BR_MoveInPlane_Acp6D_0.Parameters.Path := 2; //Y then X
			MC_BR_MoveInPlane_Acp6D_0.Execute := TRUE;
			IF MC_BR_MoveInPlane_Acp6D_0.Acknowledge THEN
				MC_BR_MoveInPlane_Acp6D_0.Execute := FALSE;
				em.substate := 3150;
			END_IF

		3150:
			em.description := 'rotationMove part 3';
			MC_BR_MoveInPlane_Acp6D_0.Shuttle := ADR(gAcp6DCtrl.Status.ShuttleInfo[3].shuttleRef);
			MC_BR_MoveInPlane_Acp6D_0.Parameters.Position.X := 0.180;
			MC_BR_MoveInPlane_Acp6D_0.Parameters.Velocity := gAcp6DCtrl.Par.Velocity;
			MC_BR_MoveInPlane_Acp6D_0.Parameters.Acceleration := gAcp6DCtrl.Par.Acceleration;
			MC_BR_MoveInPlane_Acp6D_0.Parameters.Position.Y := 0.180;
			MC_BR_MoveInPlane_Acp6D_0.Parameters.Path := 0; //direct
			MC_BR_MoveInPlane_Acp6D_0.Execute := TRUE;
			IF MC_BR_MoveInPlane_Acp6D_0.Acknowledge THEN
				MC_BR_MoveInPlane_Acp6D_0.Execute := FALSE;
				em.substate := 3160;
			END_IF

		3160:
			em.description := 'Check switch is done part 1';
			IF((gAcp6DCtrl.Status.ShuttleInfo[3].Position.X > 0.180 - MARGIN AND gAcp6DCtrl.Status.ShuttleInfo[3].Position.X < 0.180 + MARGIN) AND
				gAcp6DCtrl.Status.ShuttleInfo[3].Position.Y > 0.180 - MARGIN AND gAcp6DCtrl.Status.ShuttleInfo[3].Position.Y < 0.180 + MARGIN) THEN
				IF gAcp6DCtrl.Status.ShuttleInfo[3].State = mcACP6D_SH_STATE_IDLING THEN
					em.substate := 3170;
				END_IF
			END_IF

		3170:
			em.description := 'rotationMove part 4';
			MC_BR_MoveInPlane_Acp6D_0.Shuttle := ADR(gAcp6DCtrl.Status.ShuttleInfo[1].shuttleRef);
			MC_BR_MoveInPlane_Acp6D_0.Parameters.Position.X := 0.420;
			MC_BR_MoveInPlane_Acp6D_0.Parameters.Velocity := gAcp6DCtrl.Par.Velocity;
			MC_BR_MoveInPlane_Acp6D_0.Parameters.Acceleration := gAcp6DCtrl.Par.Acceleration;
			MC_BR_MoveInPlane_Acp6D_0.Parameters.Position.Y := 0.180;
			MC_BR_MoveInPlane_Acp6D_0.Parameters.Path := 1; //X then Y
			MC_BR_MoveInPlane_Acp6D_0.Execute := TRUE;
			IF MC_BR_MoveInPlane_Acp6D_0.Acknowledge THEN
				MC_BR_MoveInPlane_Acp6D_0.Execute := FALSE;
				em.substate := 3180;
			END_IF

		3180:
			em.description := 'Check switch is done part 2';
			IF((gAcp6DCtrl.Status.ShuttleInfo[1].Position.X > 0.420 - MARGIN AND gAcp6DCtrl.Status.ShuttleInfo[1].Position.X < 0.420 + MARGIN) AND
				gAcp6DCtrl.Status.ShuttleInfo[1].Position.Y > 0.180 - MARGIN AND gAcp6DCtrl.Status.ShuttleInfo[1].Position.Y < 0.180 + MARGIN) THEN
				IF gAcp6DCtrl.Status.ShuttleInfo[1].State = mcACP6D_SH_STATE_IDLING THEN
					em.substate := 3190;
				END_IF
			END_IF

		3190:
			em.description := 'Couple ShuttleGroup1_4';
			em.cmd.sc := FALSE;
			MC_BR_ShGroupCoupleCtrl_Acp6D_0.ShuttleGroup := shGroupShuttle1_4;
			MC_BR_ShGroupCoupleCtrl_Acp6D_0.Parameters.Option := 1; //Couple
			MC_BR_ShGroupCoupleCtrl_Acp6D_0.Execute := TRUE;
			IF MC_BR_ShGroupCoupleCtrl_Acp6D_0.Done THEN
				MC_BR_ShGroupCoupleCtrl_Acp6D_0.Execute := FALSE;
				em.substate := 3200;
			ELSIF MC_BR_ShGroupCoupleCtrl_Acp6D_0.Error THEN
				em.cmd.abort := TRUE;
			END_IF

		3200:
			em.description := 'Couple ShuttleGroup2_3';
			em.cmd.sc := FALSE;
			MC_BR_ShGroupCoupleCtrl_Acp6D_0.ShuttleGroup := shGroupShuttle2_3;
			MC_BR_ShGroupCoupleCtrl_Acp6D_0.Parameters.Option := 1; //Couple
			MC_BR_ShGroupCoupleCtrl_Acp6D_0.Execute := TRUE;
			IF MC_BR_ShGroupCoupleCtrl_Acp6D_0.Done THEN
				MC_BR_ShGroupCoupleCtrl_Acp6D_0.Execute := FALSE;
				em.substate := 3210;
			ELSIF MC_BR_ShGroupCoupleCtrl_Acp6D_0.Error THEN
				em.cmd.abort := TRUE;
			END_IF

		3210:
			em.description := 'Move right side down';
			em.cmd.sc := FALSE;
			MC_BR_MoveInPlane_Acp6D_0.Shuttle := ADR(gAcp6DCtrl.Status.ShuttleInfo[2].shuttleRef);
			MC_BR_MoveInPlane_Acp6D_0.Parameters.Position.X := 0.300;
			MC_BR_MoveInPlane_Acp6D_0.Parameters.Velocity := gAcp6DCtrl.Par.Velocity;
			MC_BR_MoveInPlane_Acp6D_0.Parameters.Acceleration := gAcp6DCtrl.Par.Acceleration;
			MC_BR_MoveInPlane_Acp6D_0.Parameters.Position.Y := 0.060;
			MC_BR_MoveInPlane_Acp6D_0.Parameters.Path := 0; //direct
			MC_BR_MoveInPlane_Acp6D_0.Execute := TRUE;
			IF MC_BR_MoveInPlane_Acp6D_0.Acknowledge THEN
				MC_BR_MoveInPlane_Acp6D_0.Execute := FALSE;
				em.substate := 3230;
			END_IF

		3230:
			em.description := 'Move group 12 of shuttle around';
			em.cmd.sc := FALSE;
			IF tempCounter >= 3 THEN
				tempCounter := 0;
				em.substate := 3250;
			ELSE
				MC_BR_MoveInPlane_Acp6D_0.Shuttle := ADR(gAcp6DCtrl.Status.ShuttleInfo[0].shuttleRef);
				MC_BR_MoveInPlane_Acp6D_0.Parameters.Position.X := 0.300;
				MC_BR_MoveInPlane_Acp6D_0.Parameters.Position.Y := 0.060;
				MC_BR_MoveInPlane_Acp6D_0.Parameters.Path := 1; //X then Y
				MC_BR_MoveInPlane_Acp6D_0.Execute := TRUE;
				IF MC_BR_MoveInPlane_Acp6D_0.Acknowledge THEN
					MC_BR_MoveInPlane_Acp6D_0.Execute := FALSE;
					em.substate := 3240;
				END_IF
			END_IF

		3240:
			em.description := 'Move group of shuttle around';
			em.cmd.sc := FALSE;
			MC_BR_MoveInPlane_Acp6D_0.Shuttle := ADR(gAcp6DCtrl.Status.ShuttleInfo[0].shuttleRef);
			MC_BR_MoveInPlane_Acp6D_0.Parameters.Position.X := 0.060;
			MC_BR_MoveInPlane_Acp6D_0.Parameters.Velocity := gAcp6DCtrl.Par.Velocity;
			MC_BR_MoveInPlane_Acp6D_0.Parameters.Acceleration := gAcp6DCtrl.Par.Acceleration;
			MC_BR_MoveInPlane_Acp6D_0.Parameters.Position.Y := 0.180;
			MC_BR_MoveInPlane_Acp6D_0.Parameters.Path := 1; //X then Y
			MC_BR_MoveInPlane_Acp6D_0.Execute := TRUE;
			IF MC_BR_MoveInPlane_Acp6D_0.Acknowledge THEN
				MC_BR_MoveInPlane_Acp6D_0.Execute := FALSE;
				tempCounter := tempCounter + 1;
				em.substate := 3230;
			END_IF

		3250:
			em.description := 'Move group 13 of shuttle around';
			em.cmd.sc := FALSE;
			IF tempCounter >= 3 THEN
				tempCounter := 0;
				em.substate := 3270;
			ELSE
				MC_BR_MoveInPlane_Acp6D_0.Shuttle := ADR(gAcp6DCtrl.Status.ShuttleInfo[2].shuttleRef);
				MC_BR_MoveInPlane_Acp6D_0.Parameters.Position.X := 0.060;
				MC_BR_MoveInPlane_Acp6D_0.Parameters.Position.Y := 0.180;
				MC_BR_MoveInPlane_Acp6D_0.Parameters.Path := 1; //X then Y
				MC_BR_MoveInPlane_Acp6D_0.Execute := TRUE;
				IF MC_BR_MoveInPlane_Acp6D_0.Acknowledge THEN
					MC_BR_MoveInPlane_Acp6D_0.Execute := FALSE;
					em.substate := 3260;
				END_IF
			END_IF

		3260:
			em.description := 'Move group of shuttle around';
			em.cmd.sc := FALSE;
			MC_BR_MoveInPlane_Acp6D_0.Shuttle := ADR(gAcp6DCtrl.Status.ShuttleInfo[2].shuttleRef);
			MC_BR_MoveInPlane_Acp6D_0.Parameters.Position.X := 0.300;
			MC_BR_MoveInPlane_Acp6D_0.Parameters.Velocity := gAcp6DCtrl.Par.Velocity;
			MC_BR_MoveInPlane_Acp6D_0.Parameters.Acceleration := gAcp6DCtrl.Par.Acceleration;
			MC_BR_MoveInPlane_Acp6D_0.Parameters.Position.Y := 0.060;
			MC_BR_MoveInPlane_Acp6D_0.Parameters.Path := 1; //X then Y
			MC_BR_MoveInPlane_Acp6D_0.Execute := TRUE;
			IF MC_BR_MoveInPlane_Acp6D_0.Acknowledge THEN
				MC_BR_MoveInPlane_Acp6D_0.Execute := FALSE;
				tempCounter := tempCounter + 1;
				em.substate := 3250;
			END_IF

		3270:
			em.cmd.sc := FALSE;
			IF((gAcp6DCtrl.Status.ShuttleInfo[2].Position.X > 0.300 - MARGIN AND gAcp6DCtrl.Status.ShuttleInfo[2].Position.X < 0.300 + MARGIN) AND
				gAcp6DCtrl.Status.ShuttleInfo[2].Position.Y > 0.060 - MARGIN AND gAcp6DCtrl.Status.ShuttleInfo[2].Position.Y < 0.060 + MARGIN) THEN
				IF gAcp6DCtrl.Status.ShuttleInfo[2].State = mcACP6D_SH_STATE_IDLING THEN
					em.substate := 3280;
				END_IF
			END_IF

		3280:
			em.description := 'Move right group up';
			em.cmd.sc := FALSE;
			MC_BR_MoveInPlane_Acp6D_0.Shuttle := ADR(gAcp6DCtrl.Status.ShuttleInfo[2].shuttleRef);
			MC_BR_MoveInPlane_Acp6D_0.Parameters.Position.X := 0.300;
			MC_BR_MoveInPlane_Acp6D_0.Parameters.Velocity := gAcp6DCtrl.Par.Velocity;
			MC_BR_MoveInPlane_Acp6D_0.Parameters.Acceleration := gAcp6DCtrl.Par.Acceleration;
			MC_BR_MoveInPlane_Acp6D_0.Parameters.Position.Y := 0.180;
			MC_BR_MoveInPlane_Acp6D_0.Parameters.Path := 0; //Direct
			MC_BR_MoveInPlane_Acp6D_0.Execute := TRUE;
			IF MC_BR_MoveInPlane_Acp6D_0.Acknowledge THEN
				MC_BR_MoveInPlane_Acp6D_0.Execute := FALSE;
				em.substate := 3290;
			END_IF

		3290:
			em.description := 'DeCouple ShuttleGroup1_4';
			em.cmd.sc := FALSE;
			MC_BR_ShGroupCoupleCtrl_Acp6D_0.ShuttleGroup := shGroupShuttle1_4;
			MC_BR_ShGroupCoupleCtrl_Acp6D_0.Parameters.Option := 0; //DeCouple
			MC_BR_ShGroupCoupleCtrl_Acp6D_0.Execute := TRUE;
			IF MC_BR_ShGroupCoupleCtrl_Acp6D_0.Done THEN
				MC_BR_ShGroupCoupleCtrl_Acp6D_0.Execute := FALSE;
				em.substate := 3300;
			ELSIF MC_BR_ShGroupCoupleCtrl_Acp6D_0.Error THEN
				em.cmd.abort := TRUE;
			END_IF

		3300:
			em.description := 'DeCouple ShuttleGroup2_3';
			em.cmd.sc := FALSE;
			MC_BR_ShGroupCoupleCtrl_Acp6D_0.ShuttleGroup := shGroupShuttle2_3;
			MC_BR_ShGroupCoupleCtrl_Acp6D_0.Parameters.Option := 0; //DeCouple
			MC_BR_ShGroupCoupleCtrl_Acp6D_0.Execute := TRUE;
			IF MC_BR_ShGroupCoupleCtrl_Acp6D_0.Done THEN
				MC_BR_ShGroupCoupleCtrl_Acp6D_0.Execute := FALSE;
				em.substate := 3310;
			ELSIF MC_BR_ShGroupCoupleCtrl_Acp6D_0.Error THEN
				em.cmd.abort := TRUE;
			END_IF

		3310:
			em.description := 'rotationMove part 1';
			MC_BR_MoveInPlane_Acp6D_0.Shuttle := ADR(gAcp6DCtrl.Status.ShuttleInfo[3].shuttleRef);
			MC_BR_MoveInPlane_Acp6D_0.Parameters.Position.X := 0.060;
			MC_BR_MoveInPlane_Acp6D_0.Parameters.Velocity := gAcp6DCtrl.Par.Velocity;
			MC_BR_MoveInPlane_Acp6D_0.Parameters.Acceleration := gAcp6DCtrl.Par.Acceleration;
			MC_BR_MoveInPlane_Acp6D_0.Parameters.Position.Y := 0.060;
			MC_BR_MoveInPlane_Acp6D_0.Parameters.Path := 2; //Y then X
			MC_BR_MoveInPlane_Acp6D_0.Execute := TRUE;
			IF MC_BR_MoveInPlane_Acp6D_0.Acknowledge THEN
				MC_BR_MoveInPlane_Acp6D_0.Execute := FALSE;
				em.substate := 3320;
			END_IF

		3320:
			em.description := 'rotationMove part 2';
			MC_BR_MoveInPlane_Acp6D_0.Shuttle := ADR(gAcp6DCtrl.Status.ShuttleInfo[1].shuttleRef);
			MC_BR_MoveInPlane_Acp6D_0.Parameters.Position.X := 0.180;
			MC_BR_MoveInPlane_Acp6D_0.Parameters.Velocity := gAcp6DCtrl.Par.Velocity;
			MC_BR_MoveInPlane_Acp6D_0.Parameters.Acceleration := gAcp6DCtrl.Par.Acceleration;
			MC_BR_MoveInPlane_Acp6D_0.Parameters.Position.Y := 0.060;
			MC_BR_MoveInPlane_Acp6D_0.Parameters.Path := 2; //Y then X
			MC_BR_MoveInPlane_Acp6D_0.Execute := TRUE;
			IF MC_BR_MoveInPlane_Acp6D_0.Acknowledge THEN
				MC_BR_MoveInPlane_Acp6D_0.Execute := FALSE;
				em.substate := 3330;
			END_IF

		3330:
			em.description := 'rotationMove part 3';
			MC_BR_MoveInPlane_Acp6D_0.Shuttle := ADR(gAcp6DCtrl.Status.ShuttleInfo[1].shuttleRef);
			MC_BR_MoveInPlane_Acp6D_0.Parameters.Position.X := 0.180;
			MC_BR_MoveInPlane_Acp6D_0.Parameters.Velocity := gAcp6DCtrl.Par.Velocity;
			MC_BR_MoveInPlane_Acp6D_0.Parameters.Acceleration := gAcp6DCtrl.Par.Acceleration;
			MC_BR_MoveInPlane_Acp6D_0.Parameters.Position.Y := 0.180;
			MC_BR_MoveInPlane_Acp6D_0.Parameters.Path := 0; //direct
			MC_BR_MoveInPlane_Acp6D_0.Execute := TRUE;
			IF MC_BR_MoveInPlane_Acp6D_0.Acknowledge THEN
				MC_BR_MoveInPlane_Acp6D_0.Execute := FALSE;
				em.substate := 3340;
			END_IF

		3340:
			IF((gAcp6DCtrl.Status.ShuttleInfo[1].Position.X > 0.180 - MARGIN AND gAcp6DCtrl.Status.ShuttleInfo[1].Position.X < 0.180 + MARGIN) AND
				gAcp6DCtrl.Status.ShuttleInfo[1].Position.Y > 0.180 - MARGIN AND gAcp6DCtrl.Status.ShuttleInfo[1].Position.Y < 0.180 + MARGIN) THEN
				IF gAcp6DCtrl.Status.ShuttleInfo[1].State = mcACP6D_SH_STATE_IDLING THEN
					em.substate := 3350;
				END_IF
			END_IF

		3350:
			em.description := 'rotationMove part 4';
			MC_BR_MoveInPlane_Acp6D_0.Shuttle := ADR(gAcp6DCtrl.Status.ShuttleInfo[3].shuttleRef);
			MC_BR_MoveInPlane_Acp6D_0.Parameters.Position.X := 0.420;
			MC_BR_MoveInPlane_Acp6D_0.Parameters.Velocity := gAcp6DCtrl.Par.Velocity;
			MC_BR_MoveInPlane_Acp6D_0.Parameters.Acceleration := gAcp6DCtrl.Par.Acceleration;
			MC_BR_MoveInPlane_Acp6D_0.Parameters.Position.Y := 0.180;
			MC_BR_MoveInPlane_Acp6D_0.Parameters.Path := 1; //X then Y
			MC_BR_MoveInPlane_Acp6D_0.Execute := TRUE;
			IF MC_BR_MoveInPlane_Acp6D_0.Acknowledge THEN
				MC_BR_MoveInPlane_Acp6D_0.Execute := FALSE;
				em.substate := 3360;
			END_IF

		3360:
			IF((gAcp6DCtrl.Status.ShuttleInfo[3].Position.X > 0.420 - MARGIN AND gAcp6DCtrl.Status.ShuttleInfo[3].Position.X < 0.420 + MARGIN) AND
				gAcp6DCtrl.Status.ShuttleInfo[3].Position.Y > 0.180 - MARGIN AND gAcp6DCtrl.Status.ShuttleInfo[3].Position.Y < 0.180 + MARGIN) THEN
				IF gAcp6DCtrl.Status.ShuttleInfo[3].State = mcACP6D_SH_STATE_IDLING THEN
					em.substate := 3030;
				END_IF
			END_IF

	END_CASE

	TON_0();

END_ACTION
```

#### conveyourStationMovement.st
```iecst
ACTION conveyorStationSetup:
	// Setup

	gWorkStations[0].par.xLocation										:= 0.180;
	gWorkStations[0].par.yLocation										:= 0.060;
	gWorkStations[0].par.nextStationSelector							:= '1';
	gWorkStations[0].par.processTime									:= ConveyorMovementWorkstation1Time;
	gWorkStations[0].par.pathRouting									:= 1;
	gWorkStations[0].par.ArcMovement									:= FALSE;
	gWorkStations[0].par.landBeforeProcess								:= FALSE;

	gWorkStations[1].par.xLocation										:= 0.420;
	gWorkStations[1].par.yLocation										:= 0.180;
	gWorkStations[1].par.nextStationSelector							:= '2';
	gWorkStations[1].par.processTime									:= ConveyorMovementWorkstation2Time;
	gWorkStations[1].par.pathRouting									:= 2;
	gWorkStations[1].par.ArcMovement									:= FALSE;
	gWorkStations[1].par.landBeforeProcess								:= FALSE;

	gWorkStations[2].par.xLocation										:= 0.060;
	gWorkStations[2].par.yLocation										:= 0.180;
	gWorkStations[2].par.nextStationSelector							:= '0';
	gWorkStations[2].par.processTime									:= 0;
	gWorkStations[2].par.pathRouting									:= 2;
	gWorkStations[2].par.ArcMovement									:= FALSE;
	gWorkStations[2].par.landBeforeProcess								:= FALSE;

	positionContainerWorkstationMov[0].initXPos							:= 0.060;
	positionContainerWorkstationMov[0].initYPos							:= 0.060;
	positionContainerWorkstationMov[1].initXPos							:= 0.180;
	positionContainerWorkstationMov[1].initYPos							:= 0.060;
	positionContainerWorkstationMov[2].initXPos							:= 0.420;
	positionContainerWorkstationMov[2].initYPos							:= 0.060;
	positionContainerWorkstationMov[3].initXPos							:= 0.420;
	positionContainerWorkstationMov[3].initYPos							:= 0.180;

	CASE em.substate OF
		9000:
			em.description := 'Move shuttle to pre pos';
			tempShuttleCounter := 0;
			MC_BR_MoveInPlaneAsync_Acp6D_0.Parameters.Acceleration := gAcp6DCtrl.Par.Acceleration;
			MC_BR_MoveInPlaneAsync_Acp6D_0.Parameters.Velocity := gAcp6DCtrl.Par.Velocity;
			FOR i := 0 TO UINT_TO_USINT(localCurrentNumShuttles-1) DO
				MC_BR_MoveInPlaneAsync_Acp6D_0.Parameters.AsyncPar[i].Shuttle := ADR(gAcp6DCtrl.Status.ShuttleInfo[i].shuttleRef);
				MC_BR_MoveInPlaneAsync_Acp6D_0.Parameters.AsyncPar[i].X := positionContainerWorkstationMov[i].initXPos;
				MC_BR_MoveInPlaneAsync_Acp6D_0.Parameters.AsyncPar[i].Y := positionContainerWorkstationMov[i].initYPos;
			END_FOR
			MC_BR_MoveInPlaneAsync_Acp6D_0.Execute := TRUE;
			IF MC_BR_MoveInPlaneAsync_Acp6D_0.Acknowledge THEN
				MC_BR_MoveInPlaneAsync_Acp6D_0.Execute := FALSE;
				em.substate := 9001;
			END_IF

		9001:
			em.description := 'Move shuttle 1 towards workstation 1';
			MC_BR_MoveInPlane_Acp6D_0.Parameters.Acceleration := gAcp6DCtrl.Par.Acceleration;
			MC_BR_MoveInPlane_Acp6D_0.Parameters.Velocity := gAcp6DCtrl.Par.Velocity;
			MC_BR_MoveInPlane_Acp6D_0.Shuttle := ADR(gAcp6DCtrl.Status.ShuttleInfo[0].shuttleRef);;
			MC_BR_MoveInPlane_Acp6D_0.Parameters.Position.X := gWorkStations[0].par.xLocation;;
			MC_BR_MoveInPlane_Acp6D_0.Parameters.Position.Y := gWorkStations[0].par.yLocation;
			MC_BR_MoveInPlane_Acp6D_0.Parameters.Path := 0; //Y then X
			MC_BR_MoveInPlane_Acp6D_0.Parameters.Mode := 0;
			MC_BR_MoveInPlane_Acp6D_0.Execute := TRUE;
			IF MC_BR_MoveInPlane_Acp6D_0.Acknowledge THEN
				MC_BR_MoveInPlane_Acp6D_0.Execute := FALSE;
				em.substate := 9002;
			END_IF

		9002:
			em.description := 'Move shuttle 3 towards workstation 2';
			MC_BR_MoveInPlane_Acp6D_0.Parameters.Acceleration := gAcp6DCtrl.Par.Acceleration;
			MC_BR_MoveInPlane_Acp6D_0.Parameters.Velocity := gAcp6DCtrl.Par.Velocity;
			MC_BR_MoveInPlane_Acp6D_0.Shuttle := ADR(gAcp6DCtrl.Status.ShuttleInfo[2].shuttleRef);;
			MC_BR_MoveInPlane_Acp6D_0.Parameters.Position.X := gWorkStations[1].par.xLocation;;
			MC_BR_MoveInPlane_Acp6D_0.Parameters.Position.Y := gWorkStations[1].par.yLocation;
			MC_BR_MoveInPlane_Acp6D_0.Parameters.Path := 0; //Y then X
			MC_BR_MoveInPlane_Acp6D_0.Parameters.Mode := 0;
			MC_BR_MoveInPlane_Acp6D_0.Execute := TRUE;
			IF MC_BR_MoveInPlane_Acp6D_0.Acknowledge THEN
				MC_BR_MoveInPlane_Acp6D_0.Execute := FALSE;
				em.substate := 9003;
			END_IF

		9003:
			// Change timer on the fly
			gWorkStations[0].par.processTime									:= ConveyorMovementWorkstation1Time;
			gWorkStations[1].par.processTime									:= ConveyorMovementWorkstation2Time;

	END_CASE

END_ACTION

ACTION conveyourStationMovement:
	// Setup
//	pWorkStations.MC_BR_MoveInPlane_Acp6D_0.Controller 					:= ADR(McAcp6DController);
//	pWorkStations.MC_BR_ShLevitation_Acp6D_0.Controller				:= ADR(McAcp6DController);
//	pWorkStations.MC_BR_MoveArcAngle_Acp6D_0.Controller					:= ADR(McAcp6DController);

	CASE cm.state OF
		// Display station at image
		//'<foreignObject x="20" y="20" width="300" height="300"><img src="Media/statusGreen.png" height="300" width="300"/>'
		//brsstrcat(ADR(showWorkStations),ADR('<foreingObject x="'));
		//brdkStrCat(ADR(showWorkStations), ADR(testDraw));
		//brdkStrCat(ADR(showWorkStations),'<foreingObject x="');

		0:
			//Check what shuttle is on top of workstation
			FOR k := 0 TO NUM_SHUTTLES DO
				IF((gAcp6DCtrl.Status.ShuttleInfo[k].Position.X > pWorkStations.par.xLocation - MARGIN AND gAcp6DCtrl.Status.ShuttleInfo[k].Position.X < pWorkStations.par.xLocation + MARGIN) AND
					gAcp6DCtrl.Status.ShuttleInfo[k].Position.Y > pWorkStations.par.yLocation - MARGIN AND gAcp6DCtrl.Status.ShuttleInfo[k].Position.Y < pWorkStations.par.yLocation + MARGIN) THEN
					IF gAcp6DCtrl.Status.ShuttleInfo[k].State = mcACP6D_SH_STATE_IDLING THEN
						pWorkStations.par.tempShuttleID := k;
						IF pWorkStations.par.landBeforeProcess THEN
							cm.state := 10;
						ELSE
							cm.state := 20;
						END_IF
					END_IF
				END_IF
			END_FOR

		10:
			//Land shuttle if reguired
			IF gAcp6DCtrl.Status.ShuttleInfo[pWorkStations.par.tempShuttleID].State = mcACP6D_SH_STATE_IDLING THEN
				pWorkStations.MC_BR_ShLevitation_Acp6D_0.Shuttle := ADR(gAcp6DCtrl.Status.ShuttleInfo[pWorkStations.par.tempShuttleID].shuttleRef);
				pWorkStations.MC_BR_ShLevitation_Acp6D_0.Parameters.Level := 0; //Land
				pWorkStations.MC_BR_ShLevitation_Acp6D_0.Parameters.Speed := 20;
				pWorkStations.MC_BR_ShLevitation_Acp6D_0.Execute := TRUE;
			END_IF
			IF pWorkStations.MC_BR_ShLevitation_Acp6D_0.Done THEN
				pWorkStations.MC_BR_ShLevitation_Acp6D_0.Execute := FALSE;
				cm.state := 15;
			END_IF

		15:
			IF gAcp6DCtrl.Status.ShuttleInfo[pWorkStations.par.tempShuttleID].State = mcACP6D_SH_STATE_LANDED THEN
				pWorkStations.TON_0.PT := t#5s;
				pWorkStations.TON_0.IN := TRUE;
				IF pWorkStations.TON_0.Q THEN
					pWorkStations.MC_BR_ShLevitation_Acp6D_0.Execute := FALSE;
					pWorkStations.TON_0.IN := FALSE;
					cm.state := 20;
				END_IF
			END_IF

		20:
			//Simulate process TON timer
			pWorkStations.TON_0.PT := REAL_TO_TIME(pWorkStations.par.processTime*1000);
			pWorkStations.TON_0.IN := TRUE;
			IF pWorkStations.TON_0.Q THEN
				pWorkStations.TON_0.IN := FALSE;
				IF pWorkStations.par.landBeforeProcess THEN
					cm.state := 30;
				ELSE
					cm.state := 40;
				END_IF
			END_IF

		30:
			//Leviate shuttle if landed before process
			pWorkStations.MC_BR_ShLevitation_Acp6D_0.Shuttle := ADR(gAcp6DCtrl.Status.ShuttleInfo[pWorkStations.par.tempShuttleID].shuttleRef);
			pWorkStations.MC_BR_ShLevitation_Acp6D_0.Parameters.Level := 1; //Leviate
			pWorkStations.MC_BR_ShLevitation_Acp6D_0.Parameters.Speed := 0;
			pWorkStations.MC_BR_ShLevitation_Acp6D_0.Execute := TRUE;
			IF pWorkStations.MC_BR_ShLevitation_Acp6D_0.Done THEN
				pWorkStations.MC_BR_ShLevitation_Acp6D_0.Execute := FALSE;
				cm.state := 40;
			END_IF

		40:
			//Move to next workstation
			IF pWorkStations.par.ArcMovement THEN
				pWorkStations.MC_BR_MoveArc_Acp6D_0.Parameters.Angular.Center.X := 0.240;
				pWorkStations.MC_BR_MoveArc_Acp6D_0.Parameters.Angular.Center.Y := 0.240;
				pWorkStations.MC_BR_MoveArc_Acp6D_0.Parameters.Acceleration := gAcp6DCtrl.Par.Acceleration;
				pWorkStations.MC_BR_MoveArc_Acp6D_0.Parameters.Velocity := gAcp6DCtrl.Par.Velocity;
				pWorkStations.MC_BR_MoveArc_Acp6D_0.Parameters.Angular.Angle := 6.28318531; //360 degrees
				pWorkStations.MC_BR_MoveArc_Acp6D_0.Parameters.Mode := 0;
				pWorkStations.MC_BR_MoveArc_Acp6D_0.Shuttle := ADR(gAcp6DCtrl.Status.ShuttleInfo[pWorkStations.par.tempShuttleID].shuttleRef);
				pWorkStations.MC_BR_MoveArc_Acp6D_0.Execute := TRUE;
				IF pWorkStations.MC_BR_MoveArc_Acp6D_0.Acknowledge THEN
					pWorkStations.status.oneshot := FALSE;
					pWorkStations.MC_BR_MoveArc_Acp6D_0.Execute := FALSE;
					cm.state := 0;
				END_IF
			ELSE
				pWorkStations.MC_BR_MoveInPlane_Acp6D_0.Shuttle := ADR(gAcp6DCtrl.Status.ShuttleInfo[pWorkStations.par.tempShuttleID].shuttleRef);
				pWorkStations.MC_BR_MoveInPlane_Acp6D_0.Parameters.Velocity := gAcp6DCtrl.Par.Velocity;
				pWorkStations.MC_BR_MoveInPlane_Acp6D_0.Parameters.Acceleration := gAcp6DCtrl.Par.Acceleration;
				pWorkStations.MC_BR_MoveInPlane_Acp6D_0.Parameters.Position.X := gWorkStations[STRING_TO_UDINT(pWorkStations.par.nextStationSelector)].par.xLocation;
				pWorkStations.MC_BR_MoveInPlane_Acp6D_0.Parameters.Position.Y := gWorkStations[STRING_TO_UDINT(pWorkStations.par.nextStationSelector)].par.yLocation;
				pWorkStations.MC_BR_MoveInPlane_Acp6D_0.Parameters.Mode := 0; //Absolute
				pWorkStations.MC_BR_MoveInPlane_Acp6D_0.Parameters.Path := pWorkStations.par.pathRouting; //0 Diagonal, 1 First X then Y, 2 First Y then X
				pWorkStations.MC_BR_MoveInPlane_Acp6D_0.Execute := TRUE;
				IF pWorkStations.MC_BR_MoveInPlane_Acp6D_0.Acknowledge THEN
					pWorkStations.status.oneshot := FALSE;
					pWorkStations.MC_BR_MoveInPlane_Acp6D_0.Execute := FALSE;
					cm.state := 0;
				END_IF
			END_IF
	END_CASE

	//Calls
	pWorkStations.MC_BR_MoveInPlane_Acp6D_0();
	pWorkStations.MC_BR_MoveArc_Acp6D_0();
	pWorkStations.MC_BR_ShLevitation_Acp6D_0();
	pWorkStations.TON_0();
	cm();

END_ACTION
```

#### workStationMovement.st
```iecst
ACTION workStationSetup:
	// Setup
	gWorkStations[0].par.xLocation										:= 0.180;
	gWorkStations[0].par.yLocation										:= 0.060;
	gWorkStations[0].par.nextStationSelector							:= '1';
	gWorkStations[0].par.processTime									:= WorkStation1MovementTimer;
	gWorkStations[0].par.pathRouting									:= 1;
	gWorkStations[0].par.landBeforeProcess								:= FALSE;
	gWorkStations[0].par.ArcMovement									:= FALSE;

	gWorkStations[1].par.xLocation										:= 0.425;
	gWorkStations[1].par.yLocation										:= 0.060;
	gWorkStations[1].par.nextStationSelector							:= '3';
	gWorkStations[1].par.processTime									:= WorkStation2And3MovementTimer;
	gWorkStations[1].par.pathRouting									:= 2;
	gWorkStations[1].par.landBeforeProcess								:= FALSE;
	gWorkStations[1].par.ArcMovement									:= FALSE;

	gWorkStations[2].par.xLocation										:= 0.425;
	gWorkStations[2].par.yLocation										:= 0.180;
	gWorkStations[2].par.nextStationSelector							:= '3';
	gWorkStations[2].par.processTime									:= WorkStation2And3MovementTimer;
	gWorkStations[2].par.pathRouting									:= 2;
	gWorkStations[2].par.landBeforeProcess								:= FALSE;
	gWorkStations[2].par.ArcMovement									:= FALSE;

	gWorkStations[3].par.xLocation										:= 0.060;
	gWorkStations[3].par.yLocation										:= 0.180;
	gWorkStations[3].par.nextStationSelector							:= '0';
	gWorkStations[3].par.processTime									:= 0;
	gWorkStations[3].par.pathRouting									:= 2;
	gWorkStations[3].par.landBeforeProcess								:= FALSE;
	gWorkStations[3].par.ArcMovement									:= FALSE;

	positionContainerWorkstationMov[0].initXPos							:= 0.060;
	positionContainerWorkstationMov[0].initYPos							:= 0.060;
	positionContainerWorkstationMov[1].initXPos							:= 0.180;
	positionContainerWorkstationMov[1].initYPos							:= 0.060;
	positionContainerWorkstationMov[2].initXPos							:= 0.420;
	positionContainerWorkstationMov[2].initYPos							:= 0.060;
	positionContainerWorkstationMov[3].initXPos							:= 0.420;
	positionContainerWorkstationMov[3].initYPos							:= 0.180;

	CASE em.substate OF
		8000:
			em.description := 'Move shuttle to pre pos';
			tempShuttleCounter := 0;
			MC_BR_MoveInPlaneAsync_Acp6D_0.Parameters.Acceleration := gAcp6DCtrl.Par.Acceleration;
			MC_BR_MoveInPlaneAsync_Acp6D_0.Parameters.Velocity := gAcp6DCtrl.Par.Velocity;
			FOR i := 0 TO UINT_TO_USINT(localCurrentNumShuttles-1) DO
				MC_BR_MoveInPlaneAsync_Acp6D_0.Parameters.AsyncPar[i].Shuttle := ADR(gAcp6DCtrl.Status.ShuttleInfo[i].shuttleRef);
				MC_BR_MoveInPlaneAsync_Acp6D_0.Parameters.AsyncPar[i].X := positionContainerWorkstationMov[i].initXPos;
				MC_BR_MoveInPlaneAsync_Acp6D_0.Parameters.AsyncPar[i].Y := positionContainerWorkstationMov[i].initYPos;
			END_FOR
			MC_BR_MoveInPlaneAsync_Acp6D_0.Execute := TRUE;
			IF MC_BR_MoveInPlaneAsync_Acp6D_0.Acknowledge THEN
				MC_BR_MoveInPlaneAsync_Acp6D_0.Execute := FALSE;
				em.substate := 8001;
			END_IF

		8001:
			em.description := 'Move shuttle 1 towards workstation 1';
			MC_BR_MoveInPlane_Acp6D_0.Parameters.Acceleration := gAcp6DCtrl.Par.Acceleration;
			MC_BR_MoveInPlane_Acp6D_0.Parameters.Velocity := gAcp6DCtrl.Par.Velocity;
			MC_BR_MoveInPlane_Acp6D_0.Shuttle := ADR(gAcp6DCtrl.Status.ShuttleInfo[0].shuttleRef);;
			MC_BR_MoveInPlane_Acp6D_0.Parameters.Position.X := gWorkStations[0].par.xLocation;;
			MC_BR_MoveInPlane_Acp6D_0.Parameters.Position.Y := gWorkStations[0].par.yLocation;
			MC_BR_MoveInPlane_Acp6D_0.Parameters.Path := 0; //Y then X
			MC_BR_MoveInPlane_Acp6D_0.Parameters.Mode := 0;
			MC_BR_MoveInPlane_Acp6D_0.Execute := TRUE;
			IF MC_BR_MoveInPlane_Acp6D_0.Acknowledge THEN
				MC_BR_MoveInPlane_Acp6D_0.Execute := FALSE;
				em.substate := 8003;
			END_IF

		8003:
			gWorkStations[0].par.processTime							:= WorkStation1MovementTimer;
			gWorkStations[1].par.processTime							:= WorkStation2And3MovementTimer;
			gWorkStations[2].par.processTime							:= WorkStation2And3MovementTimer;

	END_CASE

END_ACTION

ACTION workStationMovement:

	CASE cm.state OF
		// Display station at image
		//'<foreignObject x="20" y="20" width="300" height="300"><img src="Media/statusGreen.png" height="300" width="300"/>'
		//brsstrcat(ADR(showWorkStations),ADR('<foreingObject x="'));
		//brdkStrCat(ADR(showWorkStations), ADR(testDraw));
		//brdkStrCat(ADR(showWorkStations),'<foreingObject x="');

		0:
			//Check what shuttle is on top of workstation
			FOR k := 0 TO NUM_SHUTTLES DO
				IF((gAcp6DCtrl.Status.ShuttleInfo[k].Position.X > pWorkStations.par.xLocation - MARGIN AND gAcp6DCtrl.Status.ShuttleInfo[k].Position.X < pWorkStations.par.xLocation + MARGIN) AND
					gAcp6DCtrl.Status.ShuttleInfo[k].Position.Y > pWorkStations.par.yLocation - MARGIN AND gAcp6DCtrl.Status.ShuttleInfo[k].Position.Y < pWorkStations.par.yLocation + MARGIN) THEN
					IF gAcp6DCtrl.Status.ShuttleInfo[k].State = mcACP6D_SH_STATE_IDLING THEN
						pWorkStations.par.tempShuttleID := k;
						IF pWorkStations.par.landBeforeProcess THEN
							cm.state := 10;
						ELSE
							cm.state := 20;
						END_IF
					END_IF
				END_IF
			END_FOR

		10:
			//Land shuttle if reguired
			IF gAcp6DCtrl.Status.ShuttleInfo[pWorkStations.par.tempShuttleID].State = mcACP6D_SH_STATE_IDLING THEN
				pWorkStations.MC_BR_ShLevitation_Acp6D_0.Shuttle := ADR(gAcp6DCtrl.Status.ShuttleInfo[pWorkStations.par.tempShuttleID].shuttleRef);
				pWorkStations.MC_BR_ShLevitation_Acp6D_0.Parameters.Level := 0; //Land
				pWorkStations.MC_BR_ShLevitation_Acp6D_0.Parameters.Speed := 10;
				pWorkStations.MC_BR_ShLevitation_Acp6D_0.Execute := TRUE;
			END_IF
			IF pWorkStations.MC_BR_ShLevitation_Acp6D_0.Done THEN
				pWorkStations.MC_BR_ShLevitation_Acp6D_0.Execute := FALSE;
				cm.state := 20;
			END_IF

		20:
			//Simulate process TON timer
			pWorkStations.TON_0.PT := REAL_TO_TIME(pWorkStations.par.processTime*1000);
			pWorkStations.TON_0.IN := TRUE;

			//Chooice which position shuttle stream to watch(Vision calc)
			CASE i OF
				3: shuttleToTakePictureOf := pWorkStations.par.tempShuttleID;
			END_CASE

			IF pWorkStations.TON_0.Q THEN
				pWorkStations.TON_0.IN := FALSE;
				IF pWorkStations.par.landBeforeProcess THEN
					cm.state := 30;
				ELSE
					cm.state := 40;
				END_IF
			END_IF

		30:
			//Leviate shuttle if landed before process
			pWorkStations.MC_BR_ShLevitation_Acp6D_0.Shuttle := ADR(gAcp6DCtrl.Status.ShuttleInfo[pWorkStations.par.tempShuttleID].shuttleRef);
			pWorkStations.MC_BR_ShLevitation_Acp6D_0.Parameters.Level := 1; //Leviate
			pWorkStations.MC_BR_ShLevitation_Acp6D_0.Parameters.Speed := 10;
			pWorkStations.MC_BR_ShLevitation_Acp6D_0.Execute := TRUE;
			IF pWorkStations.MC_BR_ShLevitation_Acp6D_0.Done THEN
				pWorkStations.MC_BR_ShLevitation_Acp6D_0.Execute := FALSE;
				cm.state := 40;
			END_IF

		40:
			//Move to next workstation
			pWorkStations.MC_BR_MoveInPlane_Acp6D_0.Shuttle := ADR(gAcp6DCtrl.Status.ShuttleInfo[pWorkStations.par.tempShuttleID].shuttleRef);
			pWorkStations.MC_BR_MoveInPlane_Acp6D_0.Parameters.Velocity := gAcp6DCtrl.Par.Velocity;
			pWorkStations.MC_BR_MoveInPlane_Acp6D_0.Parameters.Acceleration := gAcp6DCtrl.Par.Acceleration;
			pWorkStations.MC_BR_MoveInPlane_Acp6D_0.Parameters.Position.X := gWorkStations[STRING_TO_UDINT(pWorkStations.par.nextStationSelector)].par.xLocation;
			pWorkStations.MC_BR_MoveInPlane_Acp6D_0.Parameters.Position.Y := gWorkStations[STRING_TO_UDINT(pWorkStations.par.nextStationSelector)].par.yLocation;
			pWorkStations.MC_BR_MoveInPlane_Acp6D_0.Parameters.Mode := 0; //Absolute
			pWorkStations.MC_BR_MoveInPlane_Acp6D_0.Parameters.Path := pWorkStations.par.pathRouting; //0 Diagonal, 1 First X then Y, 2 First Y then X
			CASE i OF
				0:
					IF pWorkStations.workstationSwitcher AND NOT pWorkStations.status.oneshot THEN
						pWorkStations.MC_BR_MoveInPlane_Acp6D_0.Parameters.Position.X := gWorkStations[STRING_TO_UDINT(pWorkStations.par.nextStationSelector)].par.xLocation;
						pWorkStations.MC_BR_MoveInPlane_Acp6D_0.Parameters.Position.Y := gWorkStations[STRING_TO_UDINT(pWorkStations.par.nextStationSelector)].par.yLocation;
						pWorkStations.status.oneshot := TRUE;
						pWorkStations.workstationSwitcher := FALSE;
					ELSIF NOT pWorkStations.workstationSwitcher AND NOT pWorkStations.status.oneshot THEN
						pWorkStations.MC_BR_MoveInPlane_Acp6D_0.Parameters.Position.X := gWorkStations[STRING_TO_UDINT(pWorkStations.par.nextStationSelector)+1].par.xLocation;
						pWorkStations.MC_BR_MoveInPlane_Acp6D_0.Parameters.Position.Y := gWorkStations[STRING_TO_UDINT(pWorkStations.par.nextStationSelector)+1].par.yLocation;
						pWorkStations.status.oneshot := TRUE;
						pWorkStations.workstationSwitcher := TRUE;
					END_IF

			END_CASE
			pWorkStations.MC_BR_MoveInPlane_Acp6D_0.Execute := TRUE;
			IF pWorkStations.MC_BR_MoveInPlane_Acp6D_0.Acknowledge THEN
				pWorkStations.status.oneshot := FALSE;
				pWorkStations.MC_BR_MoveInPlane_Acp6D_0.Execute := FALSE;
				cm.state := 0;
			END_IF
	END_CASE

	//Calls
	pWorkStations.MC_BR_MoveInPlane_Acp6D_0();
	pWorkStations.MC_BR_ShLevitation_Acp6D_0();
	pWorkStations.TON_0();
	cm();

END_ACTION
```

#### flaskProgram.st
```iecst
ACTION flaskProgramTask:
	//setup
	positionContainerFlaskProgram[0].initXPos := 0.060;
	positionContainerFlaskProgram[0].initYPos := 0.060;
	positionContainerFlaskProgram[3].initXPos := 0.060;
	positionContainerFlaskProgram[3].initYPos := 0.180;
	positionContainerFlaskProgram[2].initXPos := 0.180;
	positionContainerFlaskProgram[2].initYPos := 0.120;
	positionContainerFlaskProgram[1].initXPos := 0.360;
	positionContainerFlaskProgram[1].initYPos := 0.120;
	CASE em.substate OF
		12000:
			em.description := 'Move shuttle to pre pos';
			tempShuttleCounter := 0;
			MC_BR_MoveInPlaneAsync_Acp6D_0.Parameters.Acceleration := gAcp6DCtrl.Par.Acceleration;
			MC_BR_MoveInPlaneAsync_Acp6D_0.Parameters.Velocity := gAcp6DCtrl.Par.Velocity;
			FOR i := 0 TO UINT_TO_USINT(localCurrentNumShuttles-1) DO
				MC_BR_MoveInPlaneAsync_Acp6D_0.Parameters.AsyncPar[i].Shuttle := ADR(gAcp6DCtrl.Status.ShuttleInfo[i].shuttleRef);
				MC_BR_MoveInPlaneAsync_Acp6D_0.Parameters.AsyncPar[i].X := positionContainerFlaskProgram[i].initXPos;
				MC_BR_MoveInPlaneAsync_Acp6D_0.Parameters.AsyncPar[i].Y := positionContainerFlaskProgram[i].initYPos;
			END_FOR
			MC_BR_MoveInPlaneAsync_Acp6D_0.Execute := TRUE;
			IF MC_BR_MoveInPlaneAsync_Acp6D_0.Done THEN
				MC_BR_MoveInPlaneAsync_Acp6D_0.Execute := FALSE;
				em.substate := 12010;
			END_IF

		12010:
			em.description := 'Start circle movement on shuttle 1';
			MC_BR_MoveArc_Acp6D_0.Shuttle := ADR(gAcp6DCtrl.Status.ShuttleInfo[1].shuttleRef);
			MC_BR_MoveArc_Acp6D_0.Parameters.Option := mcACP6D_ARC_ANGULAR;
			MC_BR_MoveArc_Acp6D_0.Parameters.Acceleration := flaskProgramAcceleration;
			MC_BR_MoveArc_Acp6D_0.Parameters.Velocity := flaskProgramVelocity;
			MC_BR_MoveArc_Acp6D_0.Parameters.Angular.Center.X := 0.361;
			MC_BR_MoveArc_Acp6D_0.Parameters.Angular.Center.Y := 0.120;
			MC_BR_MoveArc_Acp6D_0.Parameters.Angular.Angle := 6283.1;
			MC_BR_MoveArc_Acp6D_0.Parameters.Mode := 0; //Abs
			MC_BR_MoveArc_Acp6D_0.Parameters.Direction := 0; //Clockwise
			MC_BR_MoveArc_Acp6D_0.Execute := TRUE;
			IF MC_BR_MoveArc_Acp6D_0.Acknowledge THEN
				MC_BR_MoveArc_Acp6D_0.Execute := FALSE;
				em.substate := 12020;
			END_IF

		12020:
			em.description := 'shuttle 1,2,3 is doing basic movement, shuttle 4 is rotation from command above';

			IF gAcp6DCtrl.Status.ShuttleInfo[1].State = mcACP6D_SH_STATE_IDLING THEN
	  			em.substate := 12030;
			END_IF

		12030:
			em.description := 'Start circle movement shuttle 1 again';
			MC_BR_MoveArc_Acp6D_0.Shuttle := ADR(gAcp6DCtrl.Status.ShuttleInfo[1].shuttleRef);
			MC_BR_MoveArc_Acp6D_0.Parameters.Option := mcACP6D_ARC_ANGULAR;
			MC_BR_MoveArc_Acp6D_0.Parameters.Acceleration := flaskProgramAcceleration;
			MC_BR_MoveArc_Acp6D_0.Parameters.Velocity := flaskProgramVelocity;
			MC_BR_MoveArc_Acp6D_0.Parameters.Angular.Center.X := 0.361;
			MC_BR_MoveArc_Acp6D_0.Parameters.Angular.Center.Y := 0.120;
			MC_BR_MoveArc_Acp6D_0.Parameters.Angular.Angle := 6283.1;
			MC_BR_MoveArc_Acp6D_0.Parameters.Mode := 0; //Abs
			MC_BR_MoveArc_Acp6D_0.Parameters.Direction := 0; //Clockwise
			MC_BR_MoveArc_Acp6D_0.Execute := TRUE;
			IF MC_BR_MoveArc_Acp6D_0.Acknowledge THEN
				MC_BR_MoveArc_Acp6D_0.Execute := FALSE;
				em.substate := 12020;
			END_IF

	END_CASE

END_ACTION
```

#### boxProgram.st
```iecst
ACTION boxProgramTask:

//	positionContainerBoxProgram[0].initXPos := 0.060;
//	positionContainerBoxProgram[0].initYPos := 0.180;
//	positionContainerBoxProgram[1].initXPos := 0.180;
//	positionContainerBoxProgram[1].initYPos := 0.060;
//	positionContainerBoxProgram[2].initXPos := 0.420;
//	positionContainerBoxProgram[2].initYPos := 0.180;
//	positionContainerBoxProgram[3].initXPos := 0.420;
//	positionContainerBoxProgram[3].initYPos := 0.060;

	CASE em.substate OF
		13000:
			em.cmd.sc := FALSE;
			em.description := 'Move shuttle to pre pos';
			positionContainerBoxProgram[0].initXPos := 0.060;
			positionContainerBoxProgram[0].initYPos := 0.180;
			positionContainerBoxProgram[1].initXPos := 0.180;
			positionContainerBoxProgram[1].initYPos := 0.060;
			positionContainerBoxProgram[2].initXPos := 0.420;
			positionContainerBoxProgram[2].initYPos := 0.180;
			positionContainerBoxProgram[3].initXPos := 0.420;
			positionContainerBoxProgram[3].initYPos := 0.060;
			tempShuttleCounter := 0;
			MC_BR_MoveInPlaneAsync_Acp6D_0.Parameters.Acceleration := gAcp6DCtrl.Par.Acceleration;
			MC_BR_MoveInPlaneAsync_Acp6D_0.Parameters.Velocity := gAcp6DCtrl.Par.Velocity;
			FOR i := 0 TO UINT_TO_USINT(localCurrentNumShuttles-1) DO
				MC_BR_MoveInPlaneAsync_Acp6D_0.Parameters.AsyncPar[i].Shuttle := ADR(gAcp6DCtrl.Status.ShuttleInfo[i].shuttleRef);
				MC_BR_MoveInPlaneAsync_Acp6D_0.Parameters.AsyncPar[i].X := positionContainerBoxProgram[i].initXPos;
				MC_BR_MoveInPlaneAsync_Acp6D_0.Parameters.AsyncPar[i].Y := positionContainerBoxProgram[i].initYPos;
			END_FOR
			MC_BR_MoveInPlaneAsync_Acp6D_0.Execute := TRUE;
			IF MC_BR_MoveInPlaneAsync_Acp6D_0.Acknowledge THEN
				MC_BR_MoveInPlaneAsync_Acp6D_0.Execute := FALSE;
				em.substate := 13010;
			END_IF

		13010:
			em.cmd.sc := FALSE;
			em.description := 'Check all shuttles are idling';
			FOR i := 0 TO NUM_SHUTTLES DO
				IF gAcp6DCtrl.Status.ShuttleInfo[i].State = mcACP6D_SH_STATE_IDLING OR gAcp6DCtrl.Status.ShuttleInfo[i].State = mcACP6D_SH_STATE_LANDED THEN
				ELSE
					EXIT;
				END_IF
			END_FOR
			IF i > NUM_SHUTTLES THEN
				em.substate := 13015;
			END_IF

		13015:
			em.description := 'Select size or start from HMI';
			IF cmdBoxProgram.smallBox OR cmdBoxProgram.bigBox THEN
				em.substate := 13020;
			ELSIF cmdBoxProgram.bottle THEN
				em.substate := 13030;
			END_IF

		13020:
			em.description := 'Move shuttle to pre pos';
			positionContainerBoxProgram[0].initXPos := 0.060;
			positionContainerBoxProgram[0].initYPos := 0.180;
			positionContainerBoxProgram[1].initXPos := 0.180;
			positionContainerBoxProgram[1].initYPos := 0.060;
			positionContainerBoxProgram[2].initXPos := 0.420;
			positionContainerBoxProgram[2].initYPos := 0.180;
			positionContainerBoxProgram[3].initXPos := 0.420;
			positionContainerBoxProgram[3].initYPos := 0.060;
			tempShuttleCounter := 0;
			MC_BR_MoveInPlaneAsync_Acp6D_0.Parameters.Acceleration := gAcp6DCtrl.Par.Acceleration;
			MC_BR_MoveInPlaneAsync_Acp6D_0.Parameters.Velocity := gAcp6DCtrl.Par.Velocity;
			FOR i := 0 TO UINT_TO_USINT(localCurrentNumShuttles-1) DO
				MC_BR_MoveInPlaneAsync_Acp6D_0.Parameters.AsyncPar[i].Shuttle := ADR(gAcp6DCtrl.Status.ShuttleInfo[i].shuttleRef);
				MC_BR_MoveInPlaneAsync_Acp6D_0.Parameters.AsyncPar[i].X := positionContainerBoxProgram[i].initXPos;
				MC_BR_MoveInPlaneAsync_Acp6D_0.Parameters.AsyncPar[i].Y := positionContainerBoxProgram[i].initYPos;
			END_FOR
			MC_BR_MoveInPlaneAsync_Acp6D_0.Execute := TRUE;
			IF MC_BR_MoveInPlaneAsync_Acp6D_0.Done THEN
				MC_BR_MoveInPlaneAsync_Acp6D_0.Execute := FALSE;
				IF cmdBoxProgram.smallBox THEN
					cmdBoxProgram.smallBox := FALSE;
					em.substate := 13100;
				ELSIF cmdBoxProgram.bigBox THEN
					cmdBoxProgram.bigBox := FALSE;
					em.substate := 13200;
				END_IF
			END_IF

		13030:
			em.description := 'Move shuttle to pre pos';
			positionContainerBoxProgram[0].initXPos := 0.180;
			positionContainerBoxProgram[0].initYPos := 0.180;
			positionContainerBoxProgram[1].initXPos := 0.060;
			positionContainerBoxProgram[1].initYPos := 0.060;
			positionContainerBoxProgram[2].initXPos := 0.420;
			positionContainerBoxProgram[2].initYPos := 0.180;
			positionContainerBoxProgram[3].initXPos := 0.420;
			positionContainerBoxProgram[3].initYPos := 0.060;
			tempShuttleCounter := 0;
			MC_BR_MoveInPlaneAsync_Acp6D_0.Parameters.Acceleration := gAcp6DCtrl.Par.Acceleration;
			MC_BR_MoveInPlaneAsync_Acp6D_0.Parameters.Velocity := gAcp6DCtrl.Par.Velocity;
			FOR i := 0 TO UINT_TO_USINT(localCurrentNumShuttles-1) DO
				MC_BR_MoveInPlaneAsync_Acp6D_0.Parameters.AsyncPar[i].Shuttle := ADR(gAcp6DCtrl.Status.ShuttleInfo[i].shuttleRef);
				MC_BR_MoveInPlaneAsync_Acp6D_0.Parameters.AsyncPar[i].X := positionContainerBoxProgram[i].initXPos;
				MC_BR_MoveInPlaneAsync_Acp6D_0.Parameters.AsyncPar[i].Y := positionContainerBoxProgram[i].initYPos;
			END_FOR
			MC_BR_MoveInPlaneAsync_Acp6D_0.Execute := TRUE;
			IF MC_BR_MoveInPlaneAsync_Acp6D_0.Done THEN
				MC_BR_MoveInPlaneAsync_Acp6D_0.Execute := FALSE;
				IF cmdBoxProgram.bottle THEN
					cmdBoxProgram.bottle := FALSE;
					em.substate := 13250;
				END_IF
			END_IF

		13100:
			em.description := 'adjust shuttle to small size box';
			MC_BR_MoveInPlane_Acp6D_0.Shuttle := ADR(gAcp6DCtrl.Status.ShuttleInfo[1].shuttleRef);
			MC_BR_MoveInPlane_Acp6D_0.Parameters.Position.X := 0.199; // at 0.180 = 80mm on x box
			MC_BR_MoveInPlane_Acp6D_0.Parameters.Position.Y := 0.085; // at 0.060 = 80mm on y box
			MC_BR_MoveInPlane_Acp6D_0.Parameters.Velocity := gAcp6DCtrl.Par.Velocity;
			MC_BR_MoveInPlane_Acp6D_0.Parameters.Acceleration := gAcp6DCtrl.Par.Acceleration;
			MC_BR_MoveInPlane_Acp6D_0.Parameters.Mode := 0;
			MC_BR_MoveInPlane_Acp6D_0.Parameters.Path := 0; //Y then X
			MC_BR_MoveInPlane_Acp6D_0.Execute := TRUE;
			IF MC_BR_MoveInPlane_Acp6D_0.Acknowledge THEN
				MC_BR_MoveInPlane_Acp6D_0.Execute := FALSE;
				em.substate := 13300;
			END_IF

		13200:
			em.description := 'adjust shuttle to big size box';
			MC_BR_MoveInPlane_Acp6D_0.Shuttle := ADR(gAcp6DCtrl.Status.ShuttleInfo[1].shuttleRef);
			MC_BR_MoveInPlane_Acp6D_0.Parameters.Position.X := 0.197; // at 0.180 = 80mm on x box
			MC_BR_MoveInPlane_Acp6D_0.Parameters.Position.Y := 0.111; // at 0.060 = 80mm on y box
			MC_BR_MoveInPlane_Acp6D_0.Parameters.Velocity := gAcp6DCtrl.Par.Velocity;
			MC_BR_MoveInPlane_Acp6D_0.Parameters.Acceleration := gAcp6DCtrl.Par.Acceleration;
			MC_BR_MoveInPlane_Acp6D_0.Parameters.Mode := 0;
			MC_BR_MoveInPlane_Acp6D_0.Parameters.Path := 0; //Y then X
			MC_BR_MoveInPlane_Acp6D_0.Execute := TRUE;
			IF MC_BR_MoveInPlane_Acp6D_0.Acknowledge THEN
				MC_BR_MoveInPlane_Acp6D_0.Execute := FALSE;
				em.substate := 13300;
			END_IF

		13250:
			em.description := 'adjust shuttle to big bottle';
			MC_BR_MoveInPlane_Acp6D_0.Shuttle := ADR(gAcp6DCtrl.Status.ShuttleInfo[0].shuttleRef);
			MC_BR_MoveInPlane_Acp6D_0.Parameters.Position.X := 0.132; // at 0.180 = 80mm on x box
			MC_BR_MoveInPlane_Acp6D_0.Parameters.Position.Y := 0.184; // at 0.060 = 80mm on y box
			MC_BR_MoveInPlane_Acp6D_0.Parameters.Velocity := gAcp6DCtrl.Par.Velocity;
			MC_BR_MoveInPlane_Acp6D_0.Parameters.Acceleration := gAcp6DCtrl.Par.Acceleration;
			MC_BR_MoveInPlane_Acp6D_0.Parameters.Mode := 0;
			MC_BR_MoveInPlane_Acp6D_0.Parameters.Path := 0; //Y then X
			MC_BR_MoveInPlane_Acp6D_0.Execute := TRUE;
			IF MC_BR_MoveInPlane_Acp6D_0.Acknowledge THEN
				MC_BR_MoveInPlane_Acp6D_0.Execute := FALSE;
				em.substate := 13310;
			END_IF

		13300:
			em.description := 'start timer';
			TON_0.PT := t#3s;
			TON_0.IN := TRUE;
			IF TON_0.Q THEN
				TON_0.IN := FALSE;
				em.substate := 13330;
			END_IF

		13310:
			em.description := 'start timer';
			TON_0.PT := t#3s;
			TON_0.IN := TRUE;
			IF TON_0.Q THEN
				TON_0.IN := FALSE;
				em.substate := 13500;
			END_IF

		13330:
			em.cmd.sc := FALSE;
			em.description := 'Couple ShuttleGroup1_2';
			MC_BR_ShGroupCoupleCtrl_Acp6D_0.ShuttleGroup := shGroupShuttle1_2;
			MC_BR_ShGroupCoupleCtrl_Acp6D_0.Parameters.Mode := 1;
			MC_BR_ShGroupCoupleCtrl_Acp6D_0.Parameters.Option := 1; //Couple
			MC_BR_ShGroupCoupleCtrl_Acp6D_0.Execute := TRUE;
			IF MC_BR_ShGroupCoupleCtrl_Acp6D_0.Done THEN
				MC_BR_ShGroupCoupleCtrl_Acp6D_0.Execute := FALSE;
				em.substate := 13340;
			END_IF

		13340:
			em.cmd.sc := FALSE;
			em.description := 'Move box around';
			MC_BR_MoveInPlane_Acp6D_0.Shuttle := ADR(gAcp6DCtrl.Status.ShuttleInfo[0].shuttleRef);;
			MC_BR_MoveInPlane_Acp6D_0.Parameters.Position.X := 0.060;
			MC_BR_MoveInPlane_Acp6D_0.Parameters.Position.Y := 0.160;
			MC_BR_MoveInPlane_Acp6D_0.Parameters.Velocity := 1;
			MC_BR_MoveInPlane_Acp6D_0.Parameters.Acceleration := 0.5;
			MC_BR_MoveInPlane_Acp6D_0.Parameters.Path := 2; //Y then X
			MC_BR_MoveInPlane_Acp6D_0.Execute := TRUE;
			IF MC_BR_MoveInPlane_Acp6D_0.Acknowledge THEN
				MC_BR_MoveInPlane_Acp6D_0.Execute := FALSE;
				em.substate := 13350;
			END_IF

		13350:
			em.cmd.sc := FALSE;
			em.description := 'Move shuttles in X Y and RZ at the same time';
			MC_BR_Move6D_Acp6D_0.Parameters.InPlane.Acceleration := 0.5;
			MC_BR_Move6D_Acp6D_0.Parameters.InPlane.Velocity := 0.14;
			MC_BR_Move6D_Acp6D_0.Shuttle := ADR(gAcp6DCtrl.Status.ShuttleInfo[0].shuttleRef);
			MC_BR_Move6D_Acp6D_0.Parameters.ShortAxis.Velocity.Rz := MC_BR_Move6D_Acp6D_0.Parameters.ShortAxis.Velocity.Ry := MC_BR_Move6D_Acp6D_0.Parameters.ShortAxis.Velocity.Rx := MC_BR_Move6D_Acp6D_0.Parameters.ShortAxis.Velocity.Z := 0.300;
			MC_BR_Move6D_Acp6D_0.Parameters.InPlane.Position.X := 0.125;
			MC_BR_Move6D_Acp6D_0.Parameters.InPlane.Position.Y := 0.180;
			MC_BR_Move6D_Acp6D_0.Parameters.ShortAxis.Position.Z := 0.001;
			MC_BR_Move6D_Acp6D_0.Parameters.ShortAxis.Position.Rx := 0;
			MC_BR_Move6D_Acp6D_0.Parameters.ShortAxis.Position.Ry := 0;
			MC_BR_Move6D_Acp6D_0.Parameters.ShortAxis.Position.Rz := 0.125;
			MC_BR_Move6D_Acp6D_0.Execute := TRUE;
			IF MC_BR_Move6D_Acp6D_0.Acknowledge THEN
				MC_BR_Move6D_Acp6D_0.Execute := FALSE;
				em.substate := 13360;
			END_IF

		13360:
			em.cmd.sc := FALSE;
			em.description := 'Move shuttles in X Y and RZ at the same time';
			MC_BR_Move6D_Acp6D_0.Parameters.InPlane.Acceleration := 0.5;
			MC_BR_Move6D_Acp6D_0.Parameters.InPlane.Velocity := 0.14;
			MC_BR_Move6D_Acp6D_0.Shuttle := ADR(gAcp6DCtrl.Status.ShuttleInfo[0].shuttleRef);
			MC_BR_Move6D_Acp6D_0.Parameters.ShortAxis.Velocity.Rz := MC_BR_Move6D_Acp6D_0.Parameters.ShortAxis.Velocity.Ry := MC_BR_Move6D_Acp6D_0.Parameters.ShortAxis.Velocity.Rx := MC_BR_Move6D_Acp6D_0.Parameters.ShortAxis.Velocity.Z := 0.300;
			MC_BR_Move6D_Acp6D_0.Parameters.InPlane.Position.X := 0.125;
			MC_BR_Move6D_Acp6D_0.Parameters.InPlane.Position.Y := 0.180;
			MC_BR_Move6D_Acp6D_0.Parameters.ShortAxis.Position.Z := 0.001;
			MC_BR_Move6D_Acp6D_0.Parameters.ShortAxis.Position.Rx := 0;
			MC_BR_Move6D_Acp6D_0.Parameters.ShortAxis.Position.Ry := 0;
			MC_BR_Move6D_Acp6D_0.Parameters.ShortAxis.Position.Rz := -0.125;
			MC_BR_Move6D_Acp6D_0.Execute := TRUE;
			IF MC_BR_Move6D_Acp6D_0.Acknowledge THEN
				MC_BR_Move6D_Acp6D_0.Execute := FALSE;
				em.substate := 13370;
			END_IF

		13370:
			em.cmd.sc := FALSE;
			em.description := 'Move shuttles in X Y and RZ at the same time';
			MC_BR_Move6D_Acp6D_0.Parameters.InPlane.Acceleration := 0.5;
			MC_BR_Move6D_Acp6D_0.Parameters.InPlane.Velocity := 0.14;
			MC_BR_Move6D_Acp6D_0.Shuttle := ADR(gAcp6DCtrl.Status.ShuttleInfo[0].shuttleRef);
			MC_BR_Move6D_Acp6D_0.Parameters.ShortAxis.Velocity.Rz := MC_BR_Move6D_Acp6D_0.Parameters.ShortAxis.Velocity.Ry := MC_BR_Move6D_Acp6D_0.Parameters.ShortAxis.Velocity.Rx := MC_BR_Move6D_Acp6D_0.Parameters.ShortAxis.Velocity.Z := 0.300;
			MC_BR_Move6D_Acp6D_0.Parameters.InPlane.Position.X := 0.060;
			MC_BR_Move6D_Acp6D_0.Parameters.InPlane.Position.Y := 0.180;
			MC_BR_Move6D_Acp6D_0.Parameters.ShortAxis.Position.Z := 0.001;
			MC_BR_Move6D_Acp6D_0.Parameters.ShortAxis.Position.Rx := 0;
			MC_BR_Move6D_Acp6D_0.Parameters.ShortAxis.Position.Ry := 0;
			MC_BR_Move6D_Acp6D_0.Parameters.ShortAxis.Position.Rz := 0.125;
			MC_BR_Move6D_Acp6D_0.Execute := TRUE;
			IF MC_BR_Move6D_Acp6D_0.Acknowledge THEN
				MC_BR_Move6D_Acp6D_0.Execute := FALSE;
				em.substate := 13380;
			END_IF

		13380:
			em.cmd.sc := FALSE;
			em.description := 'Move shuttles in X Y and RZ at the same time';
			MC_BR_Move6D_Acp6D_0.Parameters.InPlane.Acceleration := 0.5;
			MC_BR_Move6D_Acp6D_0.Parameters.InPlane.Velocity := 0.14;
			MC_BR_Move6D_Acp6D_0.Shuttle := ADR(gAcp6DCtrl.Status.ShuttleInfo[0].shuttleRef);
			MC_BR_Move6D_Acp6D_0.Parameters.ShortAxis.Velocity.Rz := MC_BR_Move6D_Acp6D_0.Parameters.ShortAxis.Velocity.Ry := MC_BR_Move6D_Acp6D_0.Parameters.ShortAxis.Velocity.Rx := MC_BR_Move6D_Acp6D_0.Parameters.ShortAxis.Velocity.Z := 0.300;
			MC_BR_Move6D_Acp6D_0.Parameters.InPlane.Position.X := 0.125;
			MC_BR_Move6D_Acp6D_0.Parameters.InPlane.Position.Y := 0.180;
			MC_BR_Move6D_Acp6D_0.Parameters.ShortAxis.Position.Z := 0.001;
			MC_BR_Move6D_Acp6D_0.Parameters.ShortAxis.Position.Rx := 0;
			MC_BR_Move6D_Acp6D_0.Parameters.ShortAxis.Position.Ry := 0;
			MC_BR_Move6D_Acp6D_0.Parameters.ShortAxis.Position.Rz := -0.125;
			MC_BR_Move6D_Acp6D_0.Execute := TRUE;
			IF MC_BR_Move6D_Acp6D_0.Acknowledge THEN
				MC_BR_Move6D_Acp6D_0.Execute := FALSE;
				em.substate := 13390;
			END_IF

		13390:
			em.cmd.sc := FALSE;
			em.description := 'Move shuttles in X Y and RZ at the same time';
			MC_BR_Move6D_Acp6D_0.Parameters.InPlane.Acceleration := 0.5;
			MC_BR_Move6D_Acp6D_0.Parameters.InPlane.Velocity := 0.14;
			MC_BR_Move6D_Acp6D_0.Shuttle := ADR(gAcp6DCtrl.Status.ShuttleInfo[0].shuttleRef);
			MC_BR_Move6D_Acp6D_0.Parameters.ShortAxis.Velocity.Rz := MC_BR_Move6D_Acp6D_0.Parameters.ShortAxis.Velocity.Ry := MC_BR_Move6D_Acp6D_0.Parameters.ShortAxis.Velocity.Rx := MC_BR_Move6D_Acp6D_0.Parameters.ShortAxis.Velocity.Z := 0.300;
			MC_BR_Move6D_Acp6D_0.Parameters.InPlane.Position.X := 0.060;
			MC_BR_Move6D_Acp6D_0.Parameters.InPlane.Position.Y := 0.180;
			MC_BR_Move6D_Acp6D_0.Parameters.ShortAxis.Position.Z := 0.001;
			MC_BR_Move6D_Acp6D_0.Parameters.ShortAxis.Position.Rx := 0;
			MC_BR_Move6D_Acp6D_0.Parameters.ShortAxis.Position.Ry := 0;
			MC_BR_Move6D_Acp6D_0.Parameters.ShortAxis.Position.Rz := 0;
			MC_BR_Move6D_Acp6D_0.Execute := TRUE;
			IF MC_BR_Move6D_Acp6D_0.Done THEN
				MC_BR_Move6D_Acp6D_0.Execute := FALSE;
				em.substate := 13400;
			END_IF

		13400:
			em.cmd.sc := FALSE;
			em.description := 'DeCouple ShuttleGroup1_2';
			MC_BR_ShGroupCoupleCtrl_Acp6D_0.ShuttleGroup := shGroupShuttle1_2;
			MC_BR_ShGroupCoupleCtrl_Acp6D_0.Parameters.Option := 0; //DeCouple
			MC_BR_ShGroupCoupleCtrl_Acp6D_0.Execute := TRUE;
			IF MC_BR_ShGroupCoupleCtrl_Acp6D_0.Done THEN
				MC_BR_ShGroupCoupleCtrl_Acp6D_0.Execute := FALSE;
				em.substate := 13010;
			END_IF

		13500:
			em.cmd.sc := FALSE;
			em.description := 'Couple ShuttleGroup1_2';
			MC_BR_ShGroupCoupleCtrl_Acp6D_0.ShuttleGroup := shGroupShuttle1_2;
			MC_BR_ShGroupCoupleCtrl_Acp6D_0.Parameters.Mode := 1;
			MC_BR_ShGroupCoupleCtrl_Acp6D_0.Parameters.Option := 1; //Couple
			MC_BR_ShGroupCoupleCtrl_Acp6D_0.Execute := TRUE;
			IF MC_BR_ShGroupCoupleCtrl_Acp6D_0.Done THEN
				MC_BR_ShGroupCoupleCtrl_Acp6D_0.Execute := FALSE;
				em.substate := 13510;
			END_IF

		13510:
			em.cmd.sc := FALSE;
			em.description := 'Move bottle around';
			MC_BR_MoveInPlane_Acp6D_0.Shuttle := ADR(gAcp6DCtrl.Status.ShuttleInfo[1].shuttleRef);;
			MC_BR_MoveInPlane_Acp6D_0.Parameters.Position.X := 0.180;
			MC_BR_MoveInPlane_Acp6D_0.Parameters.Position.Y := 0.060;
			MC_BR_MoveInPlane_Acp6D_0.Parameters.Velocity := 1;
			MC_BR_MoveInPlane_Acp6D_0.Parameters.Acceleration := 0.5;
			MC_BR_MoveInPlane_Acp6D_0.Parameters.Path := 2; //Y then X
			MC_BR_MoveInPlane_Acp6D_0.Execute := TRUE;
			IF MC_BR_MoveInPlane_Acp6D_0.Acknowledge THEN
				MC_BR_MoveInPlane_Acp6D_0.Execute := FALSE;
				em.substate := 13520;
			END_IF

		13520:
			em.cmd.sc := FALSE;
			em.description := 'Move bottle around';
			MC_BR_MoveInPlane_Acp6D_0.Shuttle := ADR(gAcp6DCtrl.Status.ShuttleInfo[1].shuttleRef);;
			MC_BR_MoveInPlane_Acp6D_0.Parameters.Position.X := 0.060;
			MC_BR_MoveInPlane_Acp6D_0.Parameters.Position.Y := 0.060;
			MC_BR_MoveInPlane_Acp6D_0.Parameters.Velocity := 1;
			MC_BR_MoveInPlane_Acp6D_0.Parameters.Acceleration := 0.5;
			MC_BR_MoveInPlane_Acp6D_0.Parameters.Path := 2; //Y then X
			MC_BR_MoveInPlane_Acp6D_0.Execute := TRUE;
			IF MC_BR_MoveInPlane_Acp6D_0.Done THEN
				MC_BR_MoveInPlane_Acp6D_0.Execute := FALSE;
				em.substate := 13400; //decouple state
			END_IF
	END_CASE

	TON_0();

END_ACTION
```
